    CONST robtarget p3347:= [[1487.1808479376136, -53.85036414256474, 992.500033578516], [0, 0, 1, 0], [0, 0, 0, 0], [9E9, 9E9, 9E9, 9E9, 9E9, 9E9]];
    CONST robtarget p3348:= [[1486.87587996053, -53.77743864899183, 992.500033578516], [0, 0, 1, 0], [0, 0, 0, 0], [9E9, 9E9, 9E9, 9E9, 9E9, 9E9]];
    CONST robtarget p3349:= [[1486.2803701551672, -53.64200512980345, 992.500033578516], [0, 0, 1, 0], [0, 0, 0, 0], [9E9, 9E9, 9E9, 9E9, 9E9, 9E9]];
    CONST robtarget p3350:= [[1486.1310585604317, -53.60921087716799, 992.500033578516], [0, 0, 1, 0], [0, 0, 0, 0], [9E9, 9E9, 9E9, 9E9, 9E9, 9E9]];
    CONST robtarget p3351:= [[1485.8708581653236, -53.549499191929584, 992.500033578516], [0, 0, 1, 0], [0, 0, 0, 0], [9E9, 9E9, 9E9, 9E9, 9E9, 9E9]];
    CONST robtarget p3352:= [[1485.4710135036546, -53.42288112586701, 992.500033578516], [0, 0, 1, 0], [0, 0, 0, 0], [9E9, 9E9, 9E9, 9E9, 9E9, 9E9]];
    CONST robtarget p3353:= [[1484.7300415279985, -53.201482726612156, 992.500033578516], [0, 0, 1, 0], [0, 0, 0, 0], [9E9, 9E9, 9E9, 9E9, 9E9, 9E9]];
    CONST robtarget p3354:= [[1484.6704427288005, -53.184901850971215, 992.500033578516], [0, 0, 1, 0], [0, 0, 0, 0], [9E9, 9E9, 9E9, 9E9, 9E9, 9E9]];
    CONST robtarget p3355:= [[1484.1819535099416, -53.02688255182427, 992.500033578516], [0, 0, 1, 0], [0, 0, 0, 0], [9E9, 9E9, 9E9, 9E9, 9E9, 9E9]];
    CONST robtarget p3356:= [[1483.924971929866, -52.957106793065265, 992.500033578516], [0, 0, 1, 0], [0, 0, 0, 0], [9E9, 9E9, 9E9, 9E9, 9E9, 9E9]];
    CONST robtarget p3357:= [[1483.840380212275, -52.9311047952195, 992.500033578516], [0, 0, 1, 0], [0, 0, 0, 0], [9E9, 9E9, 9E9, 9E9, 9E9, 9E9]];
    CONST robtarget p3358:= [[1483.1432899419212, -52.7309130716159, 992.500033578516], [0, 0, 1, 0], [0, 0, 0, 0], [9E9, 9E9, 9E9, 9E9, 9E9, 9E9]];
    CONST robtarget p3359:= [[1482.5943976643305, -52.5539516754126, 992.500033578516], [0, 0, 1, 0], [0, 0, 0, 0], [9E9, 9E9, 9E9, 9E9, 9E9, 9E9]];
    CONST robtarget p3360:= [[1482.3299474907458, -52.477779115658095, 992.500033578516], [0, 0, 1, 0], [0, 0, 0, 0], [9E9, 9E9, 9E9, 9E9, 9E9, 9E9]];
    CONST robtarget p3361:= [[1482.0010261741497, -52.38102058241606, 992.500033578516], [0, 0, 1, 0], [0, 0, 0, 0], [9E9, 9E9, 9E9, 9E9, 9E9, 9E9]];
    CONST robtarget p3362:= [[1481.5509158327018, -52.19874722975642, 992.500033578516], [0, 0, 1, 0], [0, 0, 0, 0], [9E9, 9E9, 9E9, 9E9, 9E9, 9E9]];
    CONST robtarget p3363:= [[1481.11315193246, -52.03041754687314, 992.500033578516], [0, 0, 1, 0], [0, 0, 0, 0], [9E9, 9E9, 9E9, 9E9, 9E9, 9E9]];
    CONST robtarget p3364:= [[1480.7938446633664, -51.90981571921251, 992.500033578516], [0, 0, 1, 0], [0, 0, 0, 0], [9E9, 9E9, 9E9, 9E9, 9E9, 9E9]];
    CONST robtarget p3365:= [[1480.54245378734, -51.821186668672595, 992.500033578516], [0, 0, 1, 0], [0, 0, 0, 0], [9E9, 9E9, 9E9, 9E9, 9E9, 9E9]];
    CONST robtarget p3366:= [[1480.41295095598, -51.770676335017384, 992.500033578516], [0, 0, 1, 0], [0, 0, 0, 0], [9E9, 9E9, 9E9, 9E9, 9E9, 9E9]];
    CONST robtarget p3367:= [[1480.1800345262973, -51.68403525234973, 992.500033578516], [0, 0, 1, 0], [0, 0, 0, 0], [9E9, 9E9, 9E9, 9E9, 9E9, 9E9]];
    CONST robtarget p3368:= [[1479.679579217019, -51.47045816045252, 992.500033578516], [0, 0, 1, 0], [0, 0, 0, 0], [9E9, 9E9, 9E9, 9E9, 9E9, 9E9]];
    CONST robtarget p3369:= [[1479.4242669133405, -51.37795854193503, 992.500033578516], [0, 0, 1, 0], [0, 0, 0, 0], [9E9, 9E9, 9E9, 9E9, 9E9, 9E9]];
    CONST robtarget p3370:= [[1479.11944210488, -51.27735123325023, 992.500033578516], [0, 0, 1, 0], [0, 0, 0, 0], [9E9, 9E9, 9E9, 9E9, 9E9, 9E9]];
    CONST robtarget p3371:= [[1478.9587402244965, -51.215634878753924, 992.500033578516], [0, 0, 1, 0], [0, 0, 0, 0], [9E9, 9E9, 9E9, 9E9, 9E9, 9E9]];
    CONST robtarget p3372:= [[1478.4078995703771, -51.00247068139136, 992.500033578516], [0, 0, 1, 0], [0, 0, 0, 0], [9E9, 9E9, 9E9, 9E9, 9E9, 9E9]];
    CONST robtarget p3373:= [[1477.9388565232143, -50.781502312677745, 992.500033578516], [0, 0, 1, 0], [0, 0, 0, 0], [9E9, 9E9, 9E9, 9E9, 9E9, 9E9]];
    CONST robtarget p3374:= [[1477.8276865064563, -50.735362270862616, 992.500033578516], [0, 0, 1, 0], [0, 0, 0, 0], [9E9, 9E9, 9E9, 9E9, 9E9, 9E9]];
    CONST robtarget p3375:= [[1477.1134991874192, -50.39257624403764, 992.500033578516], [0, 0, 1, 0], [0, 0, 0, 0], [9E9, 9E9, 9E9, 9E9, 9E9, 9E9]];
    CONST robtarget p3376:= [[1476.8127437004273, -50.25523619443268, 992.500033578516], [0, 0, 1, 0], [0, 0, 0, 0], [9E9, 9E9, 9E9, 9E9, 9E9, 9E9]];
    CONST robtarget p3377:= [[1476.581030580855, -50.14003244295683, 992.500033578516], [0, 0, 1, 0], [0, 0, 0, 0], [9E9, 9E9, 9E9, 9E9, 9E9, 9E9]];
    CONST robtarget p3378:= [[1476.2599962379181, -49.998280419195936, 992.500033578516], [0, 0, 1, 0], [0, 0, 0, 0], [9E9, 9E9, 9E9, 9E9, 9E9, 9E9]];
    CONST robtarget p3379:= [[1475.9104702559519, -49.840142555218655, 992.500033578516], [0, 0, 1, 0], [0, 0, 0, 0], [9E9, 9E9, 9E9, 9E9, 9E9, 9E9]];
    CONST robtarget p3380:= [[1475.4246393122305, -49.61222500336633, 992.500033578516], [0, 0, 1, 0], [0, 0, 0, 0], [9E9, 9E9, 9E9, 9E9, 9E9, 9E9]];
    CONST robtarget p3381:= [[1475.2041806503476, -49.49739674016412, 992.500033578516], [0, 0, 1, 0], [0, 0, 0, 0], [9E9, 9E9, 9E9, 9E9, 9E9, 9E9]];
    CONST robtarget p3382:= [[1474.6958711982638, -49.26805189035924, 992.500033578516], [0, 0, 1, 0], [0, 0, 0, 0], [9E9, 9E9, 9E9, 9E9, 9E9, 9E9]];
    CONST robtarget p3383:= [[1474.5346090707656, -49.18555260939496, 992.500033578516], [0, 0, 1, 0], [0, 0, 0, 0], [9E9, 9E9, 9E9, 9E9, 9E9, 9E9]];
    CONST robtarget p3384:= [[1474.4832461140786, -49.154293741446, 992.500033578516], [0, 0, 1, 0], [0, 0, 0, 0], [9E9, 9E9, 9E9, 9E9, 9E9, 9E9]];
    CONST robtarget p3385:= [[1473.9786661989287, -48.86779710482436, 992.500033578516], [0, 0, 1, 0], [0, 0, 0, 0], [9E9, 9E9, 9E9, 9E9, 9E9, 9E9]];
    CONST robtarget p3386:= [[1473.6783884368663, -48.684410713618966, 992.500033578516], [0, 0, 1, 0], [0, 0, 0, 0], [9E9, 9E9, 9E9, 9E9, 9E9, 9E9]];
    CONST robtarget p3387:= [[1473.4660175878853, -48.56892562768621, 992.500033578516], [0, 0, 1, 0], [0, 0, 0, 0], [9E9, 9E9, 9E9, 9E9, 9E9, 9E9]];
    CONST robtarget p3388:= [[1473.1610398384908, -48.40242427365542, 992.500033578516], [0, 0, 1, 0], [0, 0, 0, 0], [9E9, 9E9, 9E9, 9E9, 9E9, 9E9]];
    CONST robtarget p3389:= [[1472.8367985681707, -48.20621248412368, 992.500033578516], [0, 0, 1, 0], [0, 0, 0, 0], [9E9, 9E9, 9E9, 9E9, 9E9, 9E9]];
    CONST robtarget p3390:= [[1472.4561522390552, -48.009791772373376, 992.500033578516], [0, 0, 1, 0], [0, 0, 0, 0], [9E9, 9E9, 9E9, 9E9, 9E9, 9E9]];
    CONST robtarget p3391:= [[1472.1696380728436, -47.8383930113661, 992.500033578516], [0, 0, 1, 0], [0, 0, 0, 0], [9E9, 9E9, 9E9, 9E9, 9E9, 9E9]];
    CONST robtarget p3392:= [[1471.722110941695, -47.602916956820806, 992.500033578516], [0, 0, 1, 0], [0, 0, 0, 0], [9E9, 9E9, 9E9, 9E9, 9E9, 9E9]];
    CONST robtarget p3393:= [[1471.1098666991884, -47.258960245067954, 992.500033578516], [0, 0, 1, 0], [0, 0, 0, 0], [9E9, 9E9, 9E9, 9E9, 9E9, 9E9]];
    CONST robtarget p3394:= [[1470.720296694315, -47.00076007843536, 992.500033578516], [0, 0, 1, 0], [0, 0, 0, 0], [9E9, 9E9, 9E9, 9E9, 9E9, 9E9]];
    CONST robtarget p3395:= [[1470.35313472678, -46.74158028199264, 992.500033578516], [0, 0, 1, 0], [0, 0, 0, 0], [9E9, 9E9, 9E9, 9E9, 9E9, 9E9]];
    CONST robtarget p3396:= [[1470.1099347147267, -46.58885644915022, 992.500033578516], [0, 0, 1, 0], [0, 0, 0, 0], [9E9, 9E9, 9E9, 9E9, 9E9, 9E9]];
    CONST robtarget p3397:= [[1470.0533473815024, -46.55052435648606, 992.500033578516], [0, 0, 1, 0], [0, 0, 0, 0], [9E9, 9E9, 9E9, 9E9, 9E9, 9E9]];
    CONST robtarget p3398:= [[1469.7753241485486, -46.37599936065182, 992.500033578516], [0, 0, 1, 0], [0, 0, 0, 0], [9E9, 9E9, 9E9, 9E9, 9E9, 9E9]];
    CONST robtarget p3399:= [[1469.2259175939423, -46.010892422254685, 992.500033578516], [0, 0, 1, 0], [0, 0, 0, 0], [9E9, 9E9, 9E9, 9E9, 9E9, 9E9]];
    CONST robtarget p3400:= [[1468.7753752099943, -45.69106109718913, 992.500033578516], [0, 0, 1, 0], [0, 0, 0, 0], [9E9, 9E9, 9E9, 9E9, 9E9, 9E9]];
    CONST robtarget p3401:= [[1468.6198292044105, -45.59611312107232, 992.500033578516], [0, 0, 1, 0], [0, 0, 0, 0], [9E9, 9E9, 9E9, 9E9, 9E9, 9E9]];
    CONST robtarget p3402:= [[1468.0207049686155, -45.210283175710856, 992.500033578516], [0, 0, 1, 0], [0, 0, 0, 0], [9E9, 9E9, 9E9, 9E9, 9E9, 9E9]];
    CONST robtarget p3403:= [[1467.9426032268043, -45.16262396974101, 992.500033578516], [0, 0, 1, 0], [0, 0, 0, 0], [9E9, 9E9, 9E9, 9E9, 9E9, 9E9]];
    CONST robtarget p3404:= [[1467.7737235960665, -45.02594044699853, 992.500033578516], [0, 0, 1, 0], [0, 0, 0, 0], [9E9, 9E9, 9E9, 9E9, 9E9, 9E9]];
    CONST robtarget p3405:= [[1467.3306129242999, -44.708035159498436, 992.500033578516], [0, 0, 1, 0], [0, 0, 0, 0], [9E9, 9E9, 9E9, 9E9, 9E9, 9E9]];
    CONST robtarget p3406:= [[1466.7891375225997, -44.29104238444883, 992.500033578516], [0, 0, 1, 0], [0, 0, 0, 0], [9E9, 9E9, 9E9, 9E9, 9E9, 9E9]];
    CONST robtarget p3407:= [[1466.6930449917838, -44.218374738723874, 992.500033578516], [0, 0, 1, 0], [0, 0, 0, 0], [9E9, 9E9, 9E9, 9E9, 9E9, 9E9]];
    CONST robtarget p3408:= [[1466.6125504698477, -44.15573091450402, 992.500033578516], [0, 0, 1, 0], [0, 0, 0, 0], [9E9, 9E9, 9E9, 9E9, 9E9, 9E9]];
    CONST robtarget p3409:= [[1466.5453531413737, -44.1016987432777, 992.500033578516], [0, 0, 1, 0], [0, 0, 0, 0], [9E9, 9E9, 9E9, 9E9, 9E9, 9E9]];
    CONST robtarget p3410:= [[1466.0727069489167, -43.73594157482748, 992.500033578516], [0, 0, 1, 0], [0, 0, 0, 0], [9E9, 9E9, 9E9, 9E9, 9E9, 9E9]];
    CONST robtarget p3411:= [[1465.8449401864993, -43.55418955615802, 992.500033578516], [0, 0, 1, 0], [0, 0, 0, 0], [9E9, 9E9, 9E9, 9E9, 9E9, 9E9]];
    CONST robtarget p3412:= [[1465.4027049879091, -43.170989150472266, 992.500033578516], [0, 0, 1, 0], [0, 0, 0, 0], [9E9, 9E9, 9E9, 9E9, 9E9, 9E9]];
    CONST robtarget p3413:= [[1465.0737708983593, -42.91529482758523, 992.500033578516], [0, 0, 1, 0], [0, 0, 0, 0], [9E9, 9E9, 9E9, 9E9, 9E9, 9E9]];
    CONST robtarget p3414:= [[1464.758462542708, -42.69398236756925, 992.500033578516], [0, 0, 1, 0], [0, 0, 0, 0], [9E9, 9E9, 9E9, 9E9, 9E9, 9E9]];
    CONST robtarget p3415:= [[1464.7064575827471, -42.64949993988721, 992.500033578516], [0, 0, 1, 0], [0, 0, 0, 0], [9E9, 9E9, 9E9, 9E9, 9E9, 9E9]];
    CONST robtarget p3416:= [[1464.2049615544438, -42.25132751961473, 992.500033578516], [0, 0, 1, 0], [0, 0, 0, 0], [9E9, 9E9, 9E9, 9E9, 9E9, 9E9]];
    CONST robtarget p3417:= [[1463.630038306874, -41.732635097727126, 992.500033578516], [0, 0, 1, 0], [0, 0, 0, 0], [9E9, 9E9, 9E9, 9E9, 9E9, 9E9]];
    CONST robtarget p3418:= [[1463.4169508414868, -41.54373278258235, 992.500033578516], [0, 0, 1, 0], [0, 0, 0, 0], [9E9, 9E9, 9E9, 9E9, 9E9, 9E9]];
    CONST robtarget p3419:= [[1462.9378345294456, -41.10845872936408, 992.500033578516], [0, 0, 1, 0], [0, 0, 0, 0], [9E9, 9E9, 9E9, 9E9, 9E9, 9E9]];
    CONST robtarget p3420:= [[1462.7967031838916, -40.970170988054306, 992.500033578516], [0, 0, 1, 0], [0, 0, 0, 0], [9E9, 9E9, 9E9, 9E9, 9E9, 9E9]];
    CONST robtarget p3421:= [[1462.3892181115343, -40.624094337487456, 992.500033578516], [0, 0, 1, 0], [0, 0, 0, 0], [9E9, 9E9, 9E9, 9E9, 9E9, 9E9]];
    CONST robtarget p3422:= [[1462.1484926621697, -40.40265536007567, 992.500033578516], [0, 0, 1, 0], [0, 0, 0, 0], [9E9, 9E9, 9E9, 9E9, 9E9, 9E9]];
    CONST robtarget p3423:= [[1461.9188144316706, -40.19832888780002, 992.500033578516], [0, 0, 1, 0], [0, 0, 0, 0], [9E9, 9E9, 9E9, 9E9, 9E9, 9E9]];
    CONST robtarget p3424:= [[1461.7316067411623, -40.03100624215904, 992.500033578516], [0, 0, 1, 0], [0, 0, 0, 0], [9E9, 9E9, 9E9, 9E9, 9E9, 9E9]];
    CONST robtarget p3425:= [[1461.255703154484, -39.54403407148257, 992.500033578516], [0, 0, 1, 0], [0, 0, 0, 0], [9E9, 9E9, 9E9, 9E9, 9E9, 9E9]];
    CONST robtarget p3426:= [[1461.113593493523, -39.417810138225164, 992.500033578516], [0, 0, 1, 0], [0, 0, 0, 0], [9E9, 9E9, 9E9, 9E9, 9E9, 9E9]];
    CONST robtarget p3427:= [[1460.8243082681377, -39.117556858200075, 992.500033578516], [0, 0, 1, 0], [0, 0, 0, 0], [9E9, 9E9, 9E9, 9E9, 9E9, 9E9]];
    CONST robtarget p3428:= [[1460.6515882379688, -38.94266158745661, 992.500033578516], [0, 0, 1, 0], [0, 0, 0, 0], [9E9, 9E9, 9E9, 9E9, 9E9, 9E9]];
    CONST robtarget p3429:= [[1460.2690854199782, -38.52851516353172, 992.500033578516], [0, 0, 1, 0], [0, 0, 0, 0], [9E9, 9E9, 9E9, 9E9, 9E9, 9E9]];
    CONST robtarget p3430:= [[1460.145444752096, -38.401242774626866, 992.500033578516], [0, 0, 1, 0], [0, 0, 0, 0], [9E9, 9E9, 9E9, 9E9, 9E9, 9E9]];
    CONST robtarget p3431:= [[1459.9006997120866, -38.164320817301046, 992.500033578516], [0, 0, 1, 0], [0, 0, 0, 0], [9E9, 9E9, 9E9, 9E9, 9E9, 9E9]];
    CONST robtarget p3432:= [[1459.3337364708455, -37.572283003185476, 992.500033578516], [0, 0, 1, 0], [0, 0, 0, 0], [9E9, 9E9, 9E9, 9E9, 9E9, 9E9]];
    CONST robtarget p3433:= [[1459.0295125348634, -37.25995643815945, 992.500033578516], [0, 0, 1, 0], [0, 0, 0, 0], [9E9, 9E9, 9E9, 9E9, 9E9, 9E9]];
    CONST robtarget p3434:= [[1458.8623888247864, -37.06729815014819, 992.500033578516], [0, 0, 1, 0], [0, 0, 0, 0], [9E9, 9E9, 9E9, 9E9, 9E9, 9E9]];
    CONST robtarget p3435:= [[1458.6325053445294, -36.82857891687241, 992.500033578516], [0, 0, 1, 0], [0, 0, 0, 0], [9E9, 9E9, 9E9, 9E9, 9E9, 9E9]];
    CONST robtarget p3436:= [[1458.2543383331513, -36.37668611510166, 992.500033578516], [0, 0, 1, 0], [0, 0, 0, 0], [9E9, 9E9, 9E9, 9E9, 9E9, 9E9]];
    CONST robtarget p3437:= [[1458.027121084747, -36.0990363969632, 992.500033578516], [0, 0, 1, 0], [0, 0, 0, 0], [9E9, 9E9, 9E9, 9E9, 9E9, 9E9]];
    CONST robtarget p3438:= [[1457.606983168909, -35.57616256060792, 992.500033578516], [0, 0, 1, 0], [0, 0, 0, 0], [9E9, 9E9, 9E9, 9E9, 9E9, 9E9]];
    CONST robtarget p3439:= [[1457.4283569201107, -35.37977836110465, 992.500033578516], [0, 0, 1, 0], [0, 0, 0, 0], [9E9, 9E9, 9E9, 9E9, 9E9, 9E9]];
    CONST robtarget p3440:= [[1457.3011215960366, -35.219036477829, 992.500033578516], [0, 0, 1, 0], [0, 0, 0, 0], [9E9, 9E9, 9E9, 9E9, 9E9, 9E9]];
    CONST robtarget p3441:= [[1456.9818584121829, -34.82149399107248, 992.500033578516], [0, 0, 1, 0], [0, 0, 0, 0], [9E9, 9E9, 9E9, 9E9, 9E9, 9E9]];
    CONST robtarget p3442:= [[1456.6636166327598, -34.45580181917994, 992.500033578516], [0, 0, 1, 0], [0, 0, 0, 0], [9E9, 9E9, 9E9, 9E9, 9E9, 9E9]];
    CONST robtarget p3443:= [[1456.5323695679463, -34.29554978453682, 992.500033578516], [0, 0, 1, 0], [0, 0, 0, 0], [9E9, 9E9, 9E9, 9E9, 9E9, 9E9]];
    CONST robtarget p3444:= [[1456.3233257777242, -34.045472209657945, 992.500033578516], [0, 0, 1, 0], [0, 0, 0, 0], [9E9, 9E9, 9E9, 9E9, 9E9, 9E9]];
    CONST robtarget p3445:= [[1456.2166850399808, -33.918669267549404, 992.500033578516], [0, 0, 1, 0], [0, 0, 0, 0], [9E9, 9E9, 9E9, 9E9, 9E9, 9E9]];
    CONST robtarget p3446:= [[1456.0384938500167, -33.6602158090042, 992.500033578516], [0, 0, 1, 0], [0, 0, 0, 0], [9E9, 9E9, 9E9, 9E9, 9E9, 9E9]];
    CONST robtarget p3447:= [[1455.6908502470403, -33.169738455154864, 992.500033578516], [0, 0, 1, 0], [0, 0, 0, 0], [9E9, 9E9, 9E9, 9E9, 9E9, 9E9]];
    CONST robtarget p3448:= [[1455.5760633333898, -33.019124983816305, 992.500033578516], [0, 0, 1, 0], [0, 0, 0, 0], [9E9, 9E9, 9E9, 9E9, 9E9, 9E9]];
    CONST robtarget p3449:= [[1455.4907916846773, -32.91439129744002, 992.500033578516], [0, 0, 1, 0], [0, 0, 0, 0], [9E9, 9E9, 9E9, 9E9, 9E9, 9E9]];
    CONST robtarget p3450:= [[1455.3933901197092, -32.7724652494033, 992.500033578516], [0, 0, 1, 0], [0, 0, 0, 0], [9E9, 9E9, 9E9, 9E9, 9E9, 9E9]];
    CONST robtarget p3451:= [[1455.0836451860825, -32.34474490769912, 992.500033578516], [0, 0, 1, 0], [0, 0, 0, 0], [9E9, 9E9, 9E9, 9E9, 9E9, 9E9]];
    CONST robtarget p3452:= [[1455.0256362747637, -32.27203612221187, 992.500033578516], [0, 0, 1, 0], [0, 0, 0, 0], [9E9, 9E9, 9E9, 9E9, 9E9, 9E9]];
    CONST robtarget p3453:= [[1454.9849089470888, -32.20635720096585, 992.500033578516], [0, 0, 1, 0], [0, 0, 0, 0], [9E9, 9E9, 9E9, 9E9, 9E9, 9E9]];
    CONST robtarget p3454:= [[1454.8265637840655, -31.96721797953569, 992.500033578516], [0, 0, 1, 0], [0, 0, 0, 0], [9E9, 9E9, 9E9, 9E9, 9E9, 9E9]];
    CONST robtarget p3455:= [[1454.6476826405483, -31.70587733425765, 992.500033578516], [0, 0, 1, 0], [0, 0, 0, 0], [9E9, 9E9, 9E9, 9E9, 9E9, 9E9]];
    CONST robtarget p3456:= [[1454.2879280135612, -31.233368738334782, 992.500033578516], [0, 0, 1, 0], [0, 0, 0, 0], [9E9, 9E9, 9E9, 9E9, 9E9, 9E9]];
    CONST robtarget p3457:= [[1454.2310540800454, -31.15991131192105, 992.500033578516], [0, 0, 1, 0], [0, 0, 0, 0], [9E9, 9E9, 9E9, 9E9, 9E9, 9E9]];
    CONST robtarget p3458:= [[1454.0148081812833, -30.85863960132579, 992.500033578516], [0, 0, 1, 0], [0, 0, 0, 0], [9E9, 9E9, 9E9, 9E9, 9E9, 9E9]];
    CONST robtarget p3459:= [[1453.8782259279728, -30.658488528819916, 992.500033578516], [0, 0, 1, 0], [0, 0, 0, 0], [9E9, 9E9, 9E9, 9E9, 9E9, 9E9]];
    CONST robtarget p3460:= [[1453.7047332343661, -30.39940063569474, 992.500033578516], [0, 0, 1, 0], [0, 0, 0, 0], [9E9, 9E9, 9E9, 9E9, 9E9, 9E9]];
    CONST robtarget p3461:= [[1453.3569685886248, -29.82367260534658, 992.500033578516], [0, 0, 1, 0], [0, 0, 0, 0], [9E9, 9E9, 9E9, 9E9, 9E9, 9E9]];
    CONST robtarget p3462:= [[1453.1568211893682, -29.49263065365509, 992.500033578516], [0, 0, 1, 0], [0, 0, 0, 0], [9E9, 9E9, 9E9, 9E9, 9E9, 9E9]];
    CONST robtarget p3463:= [[1452.998690278866, -29.238377319886283, 992.500033578516], [0, 0, 1, 0], [0, 0, 0, 0], [9E9, 9E9, 9E9, 9E9, 9E9, 9E9]];
    CONST robtarget p3464:= [[1452.8914361103687, -29.0719103079496, 992.500033578516], [0, 0, 1, 0], [0, 0, 0, 0], [9E9, 9E9, 9E9, 9E9, 9E9, 9E9]];
    CONST robtarget p3465:= [[1452.710971989498, -28.76624786149432, 992.500033578516], [0, 0, 1, 0], [0, 0, 0, 0], [9E9, 9E9, 9E9, 9E9, 9E9, 9E9]];
    CONST robtarget p3466:= [[1452.4950323117525, -28.415016794012246, 992.500033578516], [0, 0, 1, 0], [0, 0, 0, 0], [9E9, 9E9, 9E9, 9E9, 9E9, 9E9]];
    CONST robtarget p3467:= [[1452.3180448544556, -28.09806084352619, 992.500033578516], [0, 0, 1, 0], [0, 0, 0, 0], [9E9, 9E9, 9E9, 9E9, 9E9, 9E9]];
    CONST robtarget p3468:= [[1452.0877233748438, -27.75046800727705, 992.500033578516], [0, 0, 1, 0], [0, 0, 0, 0], [9E9, 9E9, 9E9, 9E9, 9E9, 9E9]];
    CONST robtarget p3469:= [[1451.6606058467132, -27.04640524100038, 992.500033578516], [0, 0, 1, 0], [0, 0, 0, 0], [9E9, 9E9, 9E9, 9E9, 9E9, 9E9]];
    CONST robtarget p3470:= [[1451.5962239303992, -26.91805172162867, 992.500033578516], [0, 0, 1, 0], [0, 0, 0, 0], [9E9, 9E9, 9E9, 9E9, 9E9, 9E9]];
    CONST robtarget p3471:= [[1451.3722419824685, -26.459298942251095, 992.500033578516], [0, 0, 1, 0], [0, 0, 0, 0], [9E9, 9E9, 9E9, 9E9, 9E9, 9E9]];
    CONST robtarget p3472:= [[1451.218050210988, -26.183150546714593, 992.500033578516], [0, 0, 1, 0], [0, 0, 0, 0], [9E9, 9E9, 9E9, 9E9, 9E9, 9E9]];
    CONST robtarget p3473:= [[1451.0414892764409, -25.833096766525777, 992.500033578516], [0, 0, 1, 0], [0, 0, 0, 0], [9E9, 9E9, 9E9, 9E9, 9E9, 9E9]];
    CONST robtarget p3474:= [[1450.937388649569, -25.626608472575832, 992.500033578516], [0, 0, 1, 0], [0, 0, 0, 0], [9E9, 9E9, 9E9, 9E9, 9E9, 9E9]];
    CONST robtarget p3475:= [[1450.7626135189141, -25.29657327285075, 992.500033578516], [0, 0, 1, 0], [0, 0, 0, 0], [9E9, 9E9, 9E9, 9E9, 9E9, 9E9]];
    CONST robtarget p3476:= [[1450.5767888187597, -24.931814257633114, 992.500033578516], [0, 0, 1, 0], [0, 0, 0, 0], [9E9, 9E9, 9E9, 9E9, 9E9, 9E9]];
    CONST robtarget p3477:= [[1450.3107905505367, -24.420648005814748, 992.500033578516], [0, 0, 1, 0], [0, 0, 0, 0], [9E9, 9E9, 9E9, 9E9, 9E9, 9E9]];
    CONST robtarget p3478:= [[1450.0703210397674, -23.92574279306882, 992.500033578516], [0, 0, 1, 0], [0, 0, 0, 0], [9E9, 9E9, 9E9, 9E9, 9E9, 9E9]];
    CONST robtarget p3479:= [[1449.8480002303459, -23.493559697346946, 992.500033578516], [0, 0, 1, 0], [0, 0, 0, 0], [9E9, 9E9, 9E9, 9E9, 9E9, 9E9]];
    CONST robtarget p3480:= [[1449.8401476031047, -23.47896840986204, 992.500033578516], [0, 0, 1, 0], [0, 0, 0, 0], [9E9, 9E9, 9E9, 9E9, 9E9, 9E9]];
    CONST robtarget p3481:= [[1449.7743196513866, -23.329523112877595, 992.500033578516], [0, 0, 1, 0], [0, 0, 0, 0], [9E9, 9E9, 9E9, 9E9, 9E9, 9E9]];
    CONST robtarget p3482:= [[1449.490067459615, -22.636335832590113, 992.500033578516], [0, 0, 1, 0], [0, 0, 0, 0], [9E9, 9E9, 9E9, 9E9, 9E9, 9E9]];
    CONST robtarget p3483:= [[1449.3793270596516, -22.352133946995814, 992.500033578516], [0, 0, 1, 0], [0, 0, 0, 0], [9E9, 9E9, 9E9, 9E9, 9E9, 9E9]];
    CONST robtarget p3484:= [[1449.1617233913162, -21.89352333667363, 992.500033578516], [0, 0, 1, 0], [0, 0, 0, 0], [9E9, 9E9, 9E9, 9E9, 9E9, 9E9]];
    CONST robtarget p3485:= [[1449.1176045895998, -21.798337941021806, 992.500033578516], [0, 0, 1, 0], [0, 0, 0, 0], [9E9, 9E9, 9E9, 9E9, 9E9, 9E9]];
    CONST robtarget p3486:= [[1448.9987091221262, -21.52112647747648, 992.500033578516], [0, 0, 1, 0], [0, 0, 0, 0], [9E9, 9E9, 9E9, 9E9, 9E9, 9E9]];
    CONST robtarget p3487:= [[1448.9425986005542, -21.376342990196108, 992.500033578516], [0, 0, 1, 0], [0, 0, 0, 0], [9E9, 9E9, 9E9, 9E9, 9E9, 9E9]];
    CONST robtarget p3488:= [[1448.8290224991424, -21.113528522465906, 992.500033578516], [0, 0, 1, 0], [0, 0, 0, 0], [9E9, 9E9, 9E9, 9E9, 9E9, 9E9]];
    CONST robtarget p3489:= [[1448.7250837405568, -20.880642118370204, 992.500033578516], [0, 0, 1, 0], [0, 0, 0, 0], [9E9, 9E9, 9E9, 9E9, 9E9, 9E9]];
    CONST robtarget p3490:= [[1448.592786106188, -20.552964563670386, 992.500033578516], [0, 0, 1, 0], [0, 0, 0, 0], [9E9, 9E9, 9E9, 9E9, 9E9, 9E9]];
    CONST robtarget p3491:= [[1448.4839737748262, -20.304959229817023, 992.500033578516], [0, 0, 1, 0], [0, 0, 0, 0], [9E9, 9E9, 9E9, 9E9, 9E9, 9E9]];
    CONST robtarget p3492:= [[1448.4351233271393, -20.17234874689011, 992.500033578516], [0, 0, 1, 0], [0, 0, 0, 0], [9E9, 9E9, 9E9, 9E9, 9E9, 9E9]];
    CONST robtarget p3493:= [[1448.365696399131, -19.988516313687505, 992.500033578516], [0, 0, 1, 0], [0, 0, 0, 0], [9E9, 9E9, 9E9, 9E9, 9E9, 9E9]];
    CONST robtarget p3494:= [[1448.2067766799746, -19.62882008426967, 992.500033578516], [0, 0, 1, 0], [0, 0, 0, 0], [9E9, 9E9, 9E9, 9E9, 9E9, 9E9]];
    CONST robtarget p3495:= [[1448.1445776164344, -19.4193974113416, 992.500033578516], [0, 0, 1, 0], [0, 0, 0, 0], [9E9, 9E9, 9E9, 9E9, 9E9, 9E9]];
    CONST robtarget p3496:= [[1448.0330998698576, -19.101623794848415, 992.500033578516], [0, 0, 1, 0], [0, 0, 0, 0], [9E9, 9E9, 9E9, 9E9, 9E9, 9E9]];
    CONST robtarget p3497:= [[1447.99477449825, -18.9666175903102, 992.500033578516], [0, 0, 1, 0], [0, 0, 0, 0], [9E9, 9E9, 9E9, 9E9, 9E9, 9E9]];
    CONST robtarget p3498:= [[1447.8493306377272, -18.50273578183046, 992.500033578516], [0, 0, 1, 0], [0, 0, 0, 0], [9E9, 9E9, 9E9, 9E9, 9E9, 9E9]];
    CONST robtarget p3499:= [[1447.710091458263, -18.152457475056202, 992.500033578516], [0, 0, 1, 0], [0, 0, 0, 0], [9E9, 9E9, 9E9, 9E9, 9E9, 9E9]];
    CONST robtarget p3500:= [[1447.6300222279517, -17.927275169957845, 992.500033578516], [0, 0, 1, 0], [0, 0, 0, 0], [9E9, 9E9, 9E9, 9E9, 9E9, 9E9]];
    CONST robtarget p3501:= [[1447.4531103531453, -17.39982928374014, 992.500033578516], [0, 0, 1, 0], [0, 0, 0, 0], [9E9, 9E9, 9E9, 9E9, 9E9, 9E9]];
    CONST robtarget p3502:= [[1447.290968872516, -16.935627813711996, 992.500033578516], [0, 0, 1, 0], [0, 0, 0, 0], [9E9, 9E9, 9E9, 9E9, 9E9, 9E9]];
    CONST robtarget p3503:= [[1447.1409217422781, -16.490624161224908, 992.500033578516], [0, 0, 1, 0], [0, 0, 0, 0], [9E9, 9E9, 9E9, 9E9, 9E9, 9E9]];
    CONST robtarget p3504:= [[1447.1016279657379, -16.37617355106139, 992.500033578516], [0, 0, 1, 0], [0, 0, 0, 0], [9E9, 9E9, 9E9, 9E9, 9E9, 9E9]];
    CONST robtarget p3505:= [[1446.9486445579141, -15.93663314206443, 992.500033578516], [0, 0, 1, 0], [0, 0, 0, 0], [9E9, 9E9, 9E9, 9E9, 9E9, 9E9]];
    CONST robtarget p3506:= [[1446.8152564865, -15.401278346021833, 992.500033578516], [0, 0, 1, 0], [0, 0, 0, 0], [9E9, 9E9, 9E9, 9E9, 9E9, 9E9]];
    CONST robtarget p3507:= [[1446.7295768237227, -15.011047130391788, 992.500033578516], [0, 0, 1, 0], [0, 0, 0, 0], [9E9, 9E9, 9E9, 9E9, 9E9, 9E9]];
    CONST robtarget p3508:= [[1446.612030653954, -14.612522235073065, 992.500033578516], [0, 0, 1, 0], [0, 0, 0, 0], [9E9, 9E9, 9E9, 9E9, 9E9, 9E9]];
    CONST robtarget p3509:= [[1446.562436568088, -14.409856126046947, 992.500033578516], [0, 0, 1, 0], [0, 0, 0, 0], [9E9, 9E9, 9E9, 9E9, 9E9, 9E9]];
    CONST robtarget p3510:= [[1446.4816306006028, -14.123993635031042, 992.500033578516], [0, 0, 1, 0], [0, 0, 0, 0], [9E9, 9E9, 9E9, 9E9, 9E9, 9E9]];
    CONST robtarget p3511:= [[1446.4024648372183, -13.82132106732427, 992.500033578516], [0, 0, 1, 0], [0, 0, 0, 0], [9E9, 9E9, 9E9, 9E9, 9E9, 9E9]];
    CONST robtarget p3512:= [[1446.2581467404725, -13.273706195437228, 992.500033578516], [0, 0, 1, 0], [0, 0, 0, 0], [9E9, 9E9, 9E9, 9E9, 9E9, 9E9]];
    CONST robtarget p3513:= [[1446.138194338032, -12.802805213387018, 992.500033578516], [0, 0, 1, 0], [0, 0, 0, 0], [9E9, 9E9, 9E9, 9E9, 9E9, 9E9]];
    CONST robtarget p3514:= [[1445.938513046241, -12.033124951805334, 992.500033578516], [0, 0, 1, 0], [0, 0, 0, 0], [9E9, 9E9, 9E9, 9E9, 9E9, 9E9]];
    CONST robtarget p3515:= [[1445.923760106864, -11.954278447784198, 992.500033578516], [0, 0, 1, 0], [0, 0, 0, 0], [9E9, 9E9, 9E9, 9E9, 9E9, 9E9]];
    CONST robtarget p3516:= [[1445.8823964391556, -11.699978278644252, 992.500033578516], [0, 0, 1, 0], [0, 0, 0, 0], [9E9, 9E9, 9E9, 9E9, 9E9, 9E9]];
    CONST robtarget p3517:= [[1445.858249235026, -11.56425325097375, 992.500033578516], [0, 0, 1, 0], [0, 0, 0, 0], [9E9, 9E9, 9E9, 9E9, 9E9, 9E9]];
    CONST robtarget p3518:= [[1445.8403405666065, -11.471894054016317, 992.500033578516], [0, 0, 1, 0], [0, 0, 0, 0], [9E9, 9E9, 9E9, 9E9, 9E9, 9E9]];
    CONST robtarget p3519:= [[1445.8119897791105, -11.31890541957739, 992.500033578516], [0, 0, 1, 0], [0, 0, 0, 0], [9E9, 9E9, 9E9, 9E9, 9E9, 9E9]];
    CONST robtarget p3520:= [[1445.6586432752847, -10.571474974941466, 992.500033578516], [0, 0, 1, 0], [0, 0, 0, 0], [9E9, 9E9, 9E9, 9E9, 9E9, 9E9]];
    CONST robtarget p3521:= [[1445.6416589634534, -10.469936371774459, 992.500033578516], [0, 0, 1, 0], [0, 0, 0, 0], [9E9, 9E9, 9E9, 9E9, 9E9, 9E9]];
    CONST robtarget p3522:= [[1445.593108080078, -10.181225910298949, 992.500033578516], [0, 0, 1, 0], [0, 0, 0, 0], [9E9, 9E9, 9E9, 9E9, 9E9, 9E9]];
    CONST robtarget p3523:= [[1445.5468631117226, -9.94266718882993, 992.500033578516], [0, 0, 1, 0], [0, 0, 0, 0], [9E9, 9E9, 9E9, 9E9, 9E9, 9E9]];
    CONST robtarget p3524:= [[1445.4547342362575, -9.444153894284227, 992.500033578516], [0, 0, 1, 0], [0, 0, 0, 0], [9E9, 9E9, 9E9, 9E9, 9E9, 9E9]];
    CONST robtarget p3525:= [[1445.3714447736427, -9.010887898255525, 992.500033578516], [0, 0, 1, 0], [0, 0, 0, 0], [9E9, 9E9, 9E9, 9E9, 9E9, 9E9]];
    CONST robtarget p3526:= [[1445.2732767246098, -8.483335926873181, 992.500033578516], [0, 0, 1, 0], [0, 0, 0, 0], [9E9, 9E9, 9E9, 9E9, 9E9, 9E9]];
    CONST robtarget p3527:= [[1445.25313275983, -8.374357104724801, 992.500033578516], [0, 0, 1, 0], [0, 0, 0, 0], [9E9, 9E9, 9E9, 9E9, 9E9, 9E9]];
    CONST robtarget p3528:= [[1445.2095806999887, -7.978981630061071, 992.500033578516], [0, 0, 1, 0], [0, 0, 0, 0], [9E9, 9E9, 9E9, 9E9, 9E9, 9E9]];
    CONST robtarget p3529:= [[1445.1256311191448, -7.365424011079028, 992.500033578516], [0, 0, 1, 0], [0, 0, 0, 0], [9E9, 9E9, 9E9, 9E9, 9E9, 9E9]];
    CONST robtarget p3530:= [[1445.093389233748, -7.0807262688907, 992.500033578516], [0, 0, 1, 0], [0, 0, 0, 0], [9E9, 9E9, 9E9, 9E9, 9E9, 9E9]];
    CONST robtarget p3531:= [[1445.0770091126997, -6.938185816370513, 992.500033578516], [0, 0, 1, 0], [0, 0, 0, 0], [9E9, 9E9, 9E9, 9E9, 9E9, 9E9]];
    CONST robtarget p3532:= [[1445.0262101714134, -6.493044737196186, 992.500033578516], [0, 0, 1, 0], [0, 0, 0, 0], [9E9, 9E9, 9E9, 9E9, 9E9, 9E9]];
    CONST robtarget p3533:= [[1444.9589223996718, -5.8520673038310775, 992.500033578516], [0, 0, 1, 0], [0, 0, 0, 0], [9E9, 9E9, 9E9, 9E9, 9E9, 9E9]];
    CONST robtarget p3534:= [[1444.942957200915, -5.661944186401996, 992.500033578516], [0, 0, 1, 0], [0, 0, 0, 0], [9E9, 9E9, 9E9, 9E9, 9E9, 9E9]];
    CONST robtarget p3535:= [[1444.93858482627, -5.619251634791567, 992.500033578516], [0, 0, 1, 0], [0, 0, 0, 0], [9E9, 9E9, 9E9, 9E9, 9E9, 9E9]];
    CONST robtarget p3536:= [[1444.8754307775705, -5.054964641155507, 992.500033578516], [0, 0, 1, 0], [0, 0, 0, 0], [9E9, 9E9, 9E9, 9E9, 9E9, 9E9]];
    CONST robtarget p3537:= [[1444.8299077384686, -4.715481991021605, 992.500033578516], [0, 0, 1, 0], [0, 0, 0, 0], [9E9, 9E9, 9E9, 9E9, 9E9, 9E9]];
    CONST robtarget p3538:= [[1444.8149547608155, -4.59749911617368, 992.500033578516], [0, 0, 1, 0], [0, 0, 0, 0], [9E9, 9E9, 9E9, 9E9, 9E9, 9E9]];
    CONST robtarget p3539:= [[1444.813428207593, -4.551174813249077, 992.500033578516], [0, 0, 1, 0], [0, 0, 0, 0], [9E9, 9E9, 9E9, 9E9, 9E9, 9E9]];
    CONST robtarget p3540:= [[1444.789642708461, -4.073721118029198, 992.500033578516], [0, 0, 1, 0], [0, 0, 0, 0], [9E9, 9E9, 9E9, 9E9, 9E9, 9E9]];
    CONST robtarget p3541:= [[1444.7565988447466, -3.8072675157633995, 992.500033578516], [0, 0, 1, 0], [0, 0, 0, 0], [9E9, 9E9, 9E9, 9E9, 9E9, 9E9]];
    CONST robtarget p3542:= [[1444.7290518154543, -3.3100920942163583, 992.500033578516], [0, 0, 1, 0], [0, 0, 0, 0], [9E9, 9E9, 9E9, 9E9, 9E9, 9E9]];
    CONST robtarget p3543:= [[1444.7199692749316, -2.7495599834710163, 992.500033578516], [0, 0, 1, 0], [0, 0, 0, 0], [9E9, 9E9, 9E9, 9E9, 9E9, 9E9]];
    CONST robtarget p3544:= [[1444.719868805816, -2.621050148635959, 992.500033578516], [0, 0, 1, 0], [0, 0, 0, 0], [9E9, 9E9, 9E9, 9E9, 9E9, 9E9]];
    CONST robtarget p3545:= [[1444.7158211593426, -2.3672287977827295, 992.500033578516], [0, 0, 1, 0], [0, 0, 0, 0], [9E9, 9E9, 9E9, 9E9, 9E9, 9E9]];
    CONST robtarget p3546:= [[1444.4663405446136, -2.5286384905235195, 993.500033578516], [0, 0, 1, 0], [0, 0, 0, 0], [9E9, 9E9, 9E9, 9E9, 9E9, 9E9]];
    CONST robtarget p3547:= [[1444.4441635007622, -1.8292304588618151, 993.500033578516], [0, 0, 1, 0], [0, 0, 0, 0], [9E9, 9E9, 9E9, 9E9, 9E9, 9E9]];
    CONST robtarget p3548:= [[1444.428525603863, -1.3479255931139704, 993.500033578516], [0, 0, 1, 0], [0, 0, 0, 0], [9E9, 9E9, 9E9, 9E9, 9E9, 9E9]];
    CONST robtarget p3549:= [[1444.4174000410437, -1.0475235956110112, 993.500033578516], [0, 0, 1, 0], [0, 0, 0, 0], [9E9, 9E9, 9E9, 9E9, 9E9, 9E9]];
    CONST robtarget p3550:= [[1444.4104387675868, -0.7931788061941205, 993.500033578516], [0, 0, 1, 0], [0, 0, 0, 0], [9E9, 9E9, 9E9, 9E9, 9E9, 9E9]];
    CONST robtarget p3551:= [[1444.3908201907582, -0.5000305658536632, 993.500033578516], [0, 0, 1, 0], [0, 0, 0, 0], [9E9, 9E9, 9E9, 9E9, 9E9, 9E9]];
    CONST robtarget p3552:= [[1444.3878403243452, -0.4057105965694774, 993.500033578516], [0, 0, 1, 0], [0, 0, 0, 0], [9E9, 9E9, 9E9, 9E9, 9E9, 9E9]];
    CONST robtarget p3553:= [[1444.378812719543, 0.04115573668573802, 993.500033578516], [0, 0, 1, 0], [0, 0, 0, 0], [9E9, 9E9, 9E9, 9E9, 9E9, 9E9]];
    CONST robtarget p3554:= [[1444.3971996529272, 0.7206241421897772, 993.500033578516], [0, 0, 1, 0], [0, 0, 0, 0], [9E9, 9E9, 9E9, 9E9, 9E9, 9E9]];
    CONST robtarget p3555:= [[1444.4477772540863, 1.2756732553033174, 993.500033578516], [0, 0, 1, 0], [0, 0, 0, 0], [9E9, 9E9, 9E9, 9E9, 9E9, 9E9]];
    CONST robtarget p3556:= [[1444.470766942313, 1.6320465733553675, 993.500033578516], [0, 0, 1, 0], [0, 0, 0, 0], [9E9, 9E9, 9E9, 9E9, 9E9, 9E9]];
    CONST robtarget p3557:= [[1444.4563950861611, 2.3975781072703626, 993.500033578516], [0, 0, 1, 0], [0, 0, 0, 0], [9E9, 9E9, 9E9, 9E9, 9E9, 9E9]];
    CONST robtarget p3558:= [[1444.4969997494484, 3.4595933898866207, 993.500033578516], [0, 0, 1, 0], [0, 0, 0, 0], [9E9, 9E9, 9E9, 9E9, 9E9, 9E9]];
    CONST robtarget p3559:= [[1444.5180270622116, 3.9283626343067226, 993.500033578516], [0, 0, 1, 0], [0, 0, 0, 0], [9E9, 9E9, 9E9, 9E9, 9E9, 9E9]];
    CONST robtarget p3560:= [[1444.5320755007199, 4.180217495226117, 993.500033578516], [0, 0, 1, 0], [0, 0, 0, 0], [9E9, 9E9, 9E9, 9E9, 9E9, 9E9]];
    CONST robtarget p3561:= [[1444.5638364681504, 4.423399857044274, 993.500033578516], [0, 0, 1, 0], [0, 0, 0, 0], [9E9, 9E9, 9E9, 9E9, 9E9, 9E9]];
    CONST robtarget p3562:= [[1444.5945221601244, 4.750221146737246, 993.500033578516], [0, 0, 1, 0], [0, 0, 0, 0], [9E9, 9E9, 9E9, 9E9, 9E9, 9E9]];
    CONST robtarget p3563:= [[1444.6710804158372, 5.439612929627415, 993.500033578516], [0, 0, 1, 0], [0, 0, 0, 0], [9E9, 9E9, 9E9, 9E9, 9E9, 9E9]];
    CONST robtarget p3564:= [[1444.7059233943426, 5.756771017220018, 993.500033578516], [0, 0, 1, 0], [0, 0, 0, 0], [9E9, 9E9, 9E9, 9E9, 9E9, 9E9]];
    CONST robtarget p3565:= [[1444.7813864240288, 6.399868846253682, 993.500033578516], [0, 0, 1, 0], [0, 0, 0, 0], [9E9, 9E9, 9E9, 9E9, 9E9, 9E9]];
    CONST robtarget p3566:= [[1444.8621816645127, 7.0508629858633185, 993.500033578516], [0, 0, 1, 0], [0, 0, 0, 0], [9E9, 9E9, 9E9, 9E9, 9E9, 9E9]];
    CONST robtarget p3567:= [[1444.8862079695173, 7.395350083385225, 993.500033578516], [0, 0, 1, 0], [0, 0, 0, 0], [9E9, 9E9, 9E9, 9E9, 9E9, 9E9]];
    CONST robtarget p3568:= [[1444.9507516175283, 7.96420499306447, 993.500033578516], [0, 0, 1, 0], [0, 0, 0, 0], [9E9, 9E9, 9E9, 9E9, 9E9, 9E9]];
    CONST robtarget p3569:= [[1444.9643225395837, 8.06122200624199, 993.500033578516], [0, 0, 1, 0], [0, 0, 0, 0], [9E9, 9E9, 9E9, 9E9, 9E9, 9E9]];
    CONST robtarget p3570:= [[1445.006610153707, 8.340550046412304, 993.500033578516], [0, 0, 1, 0], [0, 0, 0, 0], [9E9, 9E9, 9E9, 9E9, 9E9, 9E9]];
    CONST robtarget p3571:= [[1445.1220891684259, 8.871981800045091, 993.500033578516], [0, 0, 1, 0], [0, 0, 0, 0], [9E9, 9E9, 9E9, 9E9, 9E9, 9E9]];
    CONST robtarget p3572:= [[1445.1453114117635, 9.006089570991321, 993.500033578516], [0, 0, 1, 0], [0, 0, 0, 0], [9E9, 9E9, 9E9, 9E9, 9E9, 9E9]];
    CONST robtarget p3573:= [[1445.2417461377509, 9.518825556421845, 993.500033578516], [0, 0, 1, 0], [0, 0, 0, 0], [9E9, 9E9, 9E9, 9E9, 9E9, 9E9]];
    CONST robtarget p3574:= [[1445.2680597934036, 9.721948112902098, 993.500033578516], [0, 0, 1, 0], [0, 0, 0, 0], [9E9, 9E9, 9E9, 9E9, 9E9, 9E9]];
    CONST robtarget p3575:= [[1445.2824501819928, 9.809116815332217, 993.500033578516], [0, 0, 1, 0], [0, 0, 0, 0], [9E9, 9E9, 9E9, 9E9, 9E9, 9E9]];
    CONST robtarget p3576:= [[1445.3158231956804, 9.985528260276467, 993.500033578516], [0, 0, 1, 0], [0, 0, 0, 0], [9E9, 9E9, 9E9, 9E9, 9E9, 9E9]];
    CONST robtarget p3577:= [[1445.4189728847298, 10.448378341408898, 993.500033578516], [0, 0, 1, 0], [0, 0, 0, 0], [9E9, 9E9, 9E9, 9E9, 9E9, 9E9]];
    CONST robtarget p3578:= [[1445.4737478292539, 10.73512926877379, 993.500033578516], [0, 0, 1, 0], [0, 0, 0, 0], [9E9, 9E9, 9E9, 9E9, 9E9, 9E9]];
    CONST robtarget p3579:= [[1445.5216283166671, 11.098489570658415, 993.500033578516], [0, 0, 1, 0], [0, 0, 0, 0], [9E9, 9E9, 9E9, 9E9, 9E9, 9E9]];
    CONST robtarget p3580:= [[1445.607844324445, 11.592914974054082, 993.500033578516], [0, 0, 1, 0], [0, 0, 0, 0], [9E9, 9E9, 9E9, 9E9, 9E9, 9E9]];
    CONST robtarget p3581:= [[1445.6465342912063, 11.782764377480092, 993.500033578516], [0, 0, 1, 0], [0, 0, 0, 0], [9E9, 9E9, 9E9, 9E9, 9E9, 9E9]];
    CONST robtarget p3582:= [[1445.6718525706506, 11.887893752436256, 993.500033578516], [0, 0, 1, 0], [0, 0, 0, 0], [9E9, 9E9, 9E9, 9E9, 9E9, 9E9]];
    CONST robtarget p3583:= [[1445.7335774426956, 12.182277578121344, 993.500033578516], [0, 0, 1, 0], [0, 0, 0, 0], [9E9, 9E9, 9E9, 9E9, 9E9, 9E9]];
    CONST robtarget p3584:= [[1445.7674247146101, 12.351660557892032, 993.500033578516], [0, 0, 1, 0], [0, 0, 0, 0], [9E9, 9E9, 9E9, 9E9, 9E9, 9E9]];
    CONST robtarget p3585:= [[1445.8384067939664, 12.60176605037536, 993.500033578516], [0, 0, 1, 0], [0, 0, 0, 0], [9E9, 9E9, 9E9, 9E9, 9E9, 9E9]];
    CONST robtarget p3586:= [[1445.9048383798565, 12.870160951727513, 993.500033578516], [0, 0, 1, 0], [0, 0, 0, 0], [9E9, 9E9, 9E9, 9E9, 9E9, 9E9]];
    CONST robtarget p3587:= [[1445.998214402726, 13.196687062136377, 993.500033578516], [0, 0, 1, 0], [0, 0, 0, 0], [9E9, 9E9, 9E9, 9E9, 9E9, 9E9]];
    CONST robtarget p3588:= [[1446.0463947546464, 13.402721705057857, 993.500033578516], [0, 0, 1, 0], [0, 0, 0, 0], [9E9, 9E9, 9E9, 9E9, 9E9, 9E9]];
    CONST robtarget p3589:= [[1446.1997438178155, 13.911869805080471, 993.500033578516], [0, 0, 1, 0], [0, 0, 0, 0], [9E9, 9E9, 9E9, 9E9, 9E9, 9E9]];
    CONST robtarget p3590:= [[1446.2762629473796, 14.245535715658704, 993.500033578516], [0, 0, 1, 0], [0, 0, 0, 0], [9E9, 9E9, 9E9, 9E9, 9E9, 9E9]];
    CONST robtarget p3591:= [[1446.3950136263534, 14.746056132894921, 993.500033578516], [0, 0, 1, 0], [0, 0, 0, 0], [9E9, 9E9, 9E9, 9E9, 9E9, 9E9]];
    CONST robtarget p3592:= [[1446.4997506124657, 15.08648877165038, 993.500033578516], [0, 0, 1, 0], [0, 0, 0, 0], [9E9, 9E9, 9E9, 9E9, 9E9, 9E9]];
    CONST robtarget p3593:= [[1446.575430012217, 15.404500244985172, 993.500033578516], [0, 0, 1, 0], [0, 0, 0, 0], [9E9, 9E9, 9E9, 9E9, 9E9, 9E9]];
    CONST robtarget p3594:= [[1446.6335092628235, 15.643524526965578, 993.500033578516], [0, 0, 1, 0], [0, 0, 0, 0], [9E9, 9E9, 9E9, 9E9, 9E9, 9E9]];
    CONST robtarget p3595:= [[1446.7031807526187, 15.890349156086373, 993.500033578516], [0, 0, 1, 0], [0, 0, 0, 0], [9E9, 9E9, 9E9, 9E9, 9E9, 9E9]];
    CONST robtarget p3596:= [[1446.749482642183, 16.077923135514027, 993.500033578516], [0, 0, 1, 0], [0, 0, 0, 0], [9E9, 9E9, 9E9, 9E9, 9E9, 9E9]];
    CONST robtarget p3597:= [[1446.8114590668554, 16.239465660020116, 993.500033578516], [0, 0, 1, 0], [0, 0, 0, 0], [9E9, 9E9, 9E9, 9E9, 9E9, 9E9]];
    CONST robtarget p3598:= [[1446.9146230357603, 16.53767565578663, 993.500033578516], [0, 0, 1, 0], [0, 0, 0, 0], [9E9, 9E9, 9E9, 9E9, 9E9, 9E9]];
    CONST robtarget p3599:= [[1446.963168670901, 16.66854774085074, 993.500033578516], [0, 0, 1, 0], [0, 0, 0, 0], [9E9, 9E9, 9E9, 9E9, 9E9, 9E9]];
    CONST robtarget p3600:= [[1446.9900299425199, 16.7425065795654, 993.500033578516], [0, 0, 1, 0], [0, 0, 0, 0], [9E9, 9E9, 9E9, 9E9, 9E9, 9E9]];
    CONST robtarget p3601:= [[1447.115491548474, 17.139664548150634, 993.500033578516], [0, 0, 1, 0], [0, 0, 0, 0], [9E9, 9E9, 9E9, 9E9, 9E9, 9E9]];
    CONST robtarget p3602:= [[1447.1389508457935, 17.22157378939157, 993.500033578516], [0, 0, 1, 0], [0, 0, 0, 0], [9E9, 9E9, 9E9, 9E9, 9E9, 9E9]];
    CONST robtarget p3603:= [[1447.291425586272, 17.63782814210286, 993.500033578516], [0, 0, 1, 0], [0, 0, 0, 0], [9E9, 9E9, 9E9, 9E9, 9E9, 9E9]];
    CONST robtarget p3604:= [[1447.3899407387735, 17.946634912413217, 993.500033578516], [0, 0, 1, 0], [0, 0, 0, 0], [9E9, 9E9, 9E9, 9E9, 9E9, 9E9]];
    CONST robtarget p3605:= [[1447.4383730731518, 18.098735357092124, 993.500033578516], [0, 0, 1, 0], [0, 0, 0, 0], [9E9, 9E9, 9E9, 9E9, 9E9, 9E9]];
    CONST robtarget p3606:= [[1447.565649674499, 18.435373736468506, 993.500033578516], [0, 0, 1, 0], [0, 0, 0, 0], [9E9, 9E9, 9E9, 9E9, 9E9, 9E9]];
    CONST robtarget p3607:= [[1447.6759540256755, 18.77435899441376, 993.500033578516], [0, 0, 1, 0], [0, 0, 0, 0], [9E9, 9E9, 9E9, 9E9, 9E9, 9E9]];
    CONST robtarget p3608:= [[1447.7180461341088, 18.8951522215865, 993.500033578516], [0, 0, 1, 0], [0, 0, 0, 0], [9E9, 9E9, 9E9, 9E9, 9E9, 9E9]];
    CONST robtarget p3609:= [[1447.9714600987909, 19.647451168715463, 993.500033578516], [0, 0, 1, 0], [0, 0, 0, 0], [9E9, 9E9, 9E9, 9E9, 9E9, 9E9]];
    CONST robtarget p3610:= [[1448.0516488997882, 19.887886445543487, 993.500033578516], [0, 0, 1, 0], [0, 0, 0, 0], [9E9, 9E9, 9E9, 9E9, 9E9, 9E9]];
    CONST robtarget p3611:= [[1448.0855779105252, 19.96749282121084, 993.500033578516], [0, 0, 1, 0], [0, 0, 0, 0], [9E9, 9E9, 9E9, 9E9, 9E9, 9E9]];
    CONST robtarget p3612:= [[1448.231774689219, 20.30060637761079, 993.500033578516], [0, 0, 1, 0], [0, 0, 0, 0], [9E9, 9E9, 9E9, 9E9, 9E9, 9E9]];
    CONST robtarget p3613:= [[1448.4249949476991, 20.771547217307756, 993.500033578516], [0, 0, 1, 0], [0, 0, 0, 0], [9E9, 9E9, 9E9, 9E9, 9E9, 9E9]];
    CONST robtarget p3614:= [[1448.4871546623035, 20.91339688820048, 993.500033578516], [0, 0, 1, 0], [0, 0, 0, 0], [9E9, 9E9, 9E9, 9E9, 9E9, 9E9]];
    CONST robtarget p3615:= [[1448.6708299281984, 21.346755088002624, 993.500033578516], [0, 0, 1, 0], [0, 0, 0, 0], [9E9, 9E9, 9E9, 9E9, 9E9, 9E9]];
    CONST robtarget p3616:= [[1448.9039866989838, 21.897020387037188, 993.500033578516], [0, 0, 1, 0], [0, 0, 0, 0], [9E9, 9E9, 9E9, 9E9, 9E9, 9E9]];
    CONST robtarget p3617:= [[1449.0517279863207, 22.251302004122692, 993.500033578516], [0, 0, 1, 0], [0, 0, 0, 0], [9E9, 9E9, 9E9, 9E9, 9E9, 9E9]];
    CONST robtarget p3618:= [[1449.2393358217416, 22.672920594804765, 993.500033578516], [0, 0, 1, 0], [0, 0, 0, 0], [9E9, 9E9, 9E9, 9E9, 9E9, 9E9]];
    CONST robtarget p3619:= [[1449.320061751566, 22.874129914388362, 993.500033578516], [0, 0, 1, 0], [0, 0, 0, 0], [9E9, 9E9, 9E9, 9E9, 9E9, 9E9]];
    CONST robtarget p3620:= [[1449.4529423222662, 23.175128115541014, 993.500033578516], [0, 0, 1, 0], [0, 0, 0, 0], [9E9, 9E9, 9E9, 9E9, 9E9, 9E9]];
    CONST robtarget p3621:= [[1449.4945941390156, 23.27668269252105, 993.500033578516], [0, 0, 1, 0], [0, 0, 0, 0], [9E9, 9E9, 9E9, 9E9, 9E9, 9E9]];
    CONST robtarget p3622:= [[1449.6231415702, 23.594832616201174, 993.500033578516], [0, 0, 1, 0], [0, 0, 0, 0], [9E9, 9E9, 9E9, 9E9, 9E9, 9E9]];
    CONST robtarget p3623:= [[1449.793827718006, 23.92004763440994, 993.500033578516], [0, 0, 1, 0], [0, 0, 0, 0], [9E9, 9E9, 9E9, 9E9, 9E9, 9E9]];
    CONST robtarget p3624:= [[1450.1388550638192, 24.583329948521325, 993.500033578516], [0, 0, 1, 0], [0, 0, 0, 0], [9E9, 9E9, 9E9, 9E9, 9E9, 9E9]];
    CONST robtarget p3625:= [[1450.2106914258848, 24.731601716591214, 993.500033578516], [0, 0, 1, 0], [0, 0, 0, 0], [9E9, 9E9, 9E9, 9E9, 9E9, 9E9]];
    CONST robtarget p3626:= [[1450.3869424847544, 25.078361949898607, 993.500033578516], [0, 0, 1, 0], [0, 0, 0, 0], [9E9, 9E9, 9E9, 9E9, 9E9, 9E9]];
    CONST robtarget p3627:= [[1450.4483093517806, 25.20364262778959, 993.500033578516], [0, 0, 1, 0], [0, 0, 0, 0], [9E9, 9E9, 9E9, 9E9, 9E9, 9E9]];
    CONST robtarget p3628:= [[1450.5592616233278, 25.41385635248946, 993.500033578516], [0, 0, 1, 0], [0, 0, 0, 0], [9E9, 9E9, 9E9, 9E9, 9E9, 9E9]];
    CONST robtarget p3629:= [[1450.6662676315955, 25.612184080744953, 993.500033578516], [0, 0, 1, 0], [0, 0, 0, 0], [9E9, 9E9, 9E9, 9E9, 9E9, 9E9]];
    CONST robtarget p3630:= [[1451.0725475657875, 26.41672561044352, 993.500033578516], [0, 0, 1, 0], [0, 0, 0, 0], [9E9, 9E9, 9E9, 9E9, 9E9, 9E9]];
    CONST robtarget p3631:= [[1451.452446368639, 27.11184788510795, 993.500033578516], [0, 0, 1, 0], [0, 0, 0, 0], [9E9, 9E9, 9E9, 9E9, 9E9, 9E9]];
    CONST robtarget p3632:= [[1451.5658213058541, 27.300875817009157, 993.500033578516], [0, 0, 1, 0], [0, 0, 0, 0], [9E9, 9E9, 9E9, 9E9, 9E9, 9E9]];
    CONST robtarget p3633:= [[1451.8239453307413, 27.775893752806056, 993.500033578516], [0, 0, 1, 0], [0, 0, 0, 0], [9E9, 9E9, 9E9, 9E9, 9E9, 9E9]];
    CONST robtarget p3634:= [[1451.8673058367597, 27.84268994217308, 993.500033578516], [0, 0, 1, 0], [0, 0, 0, 0], [9E9, 9E9, 9E9, 9E9, 9E9, 9E9]];
    CONST robtarget p3635:= [[1452.0289371690612, 28.094260015711797, 993.500033578516], [0, 0, 1, 0], [0, 0, 0, 0], [9E9, 9E9, 9E9, 9E9, 9E9, 9E9]];
    CONST robtarget p3636:= [[1452.207799621548, 28.38239021182298, 993.500033578516], [0, 0, 1, 0], [0, 0, 0, 0], [9E9, 9E9, 9E9, 9E9, 9E9, 9E9]];
    CONST robtarget p3637:= [[1452.2330896153153, 28.422617835947307, 993.500033578516], [0, 0, 1, 0], [0, 0, 0, 0], [9E9, 9E9, 9E9, 9E9, 9E9, 9E9]];
    CONST robtarget p3638:= [[1452.4619878307856, 28.792979689955587, 993.500033578516], [0, 0, 1, 0], [0, 0, 0, 0], [9E9, 9E9, 9E9, 9E9, 9E9, 9E9]];
    CONST robtarget p3639:= [[1452.533597025428, 28.905481381419136, 993.500033578516], [0, 0, 1, 0], [0, 0, 0, 0], [9E9, 9E9, 9E9, 9E9, 9E9, 9E9]];
    CONST robtarget p3640:= [[1452.8313620688805, 29.420512473147213, 993.500033578516], [0, 0, 1, 0], [0, 0, 0, 0], [9E9, 9E9, 9E9, 9E9, 9E9, 9E9]];
    CONST robtarget p3641:= [[1452.9340043735583, 29.58841246191679, 993.500033578516], [0, 0, 1, 0], [0, 0, 0, 0], [9E9, 9E9, 9E9, 9E9, 9E9, 9E9]];
    CONST robtarget p3642:= [[1453.0994544901425, 29.860442423281413, 993.500033578516], [0, 0, 1, 0], [0, 0, 0, 0], [9E9, 9E9, 9E9, 9E9, 9E9, 9E9]];
    CONST robtarget p3643:= [[1453.161528064843, 29.967482417793306, 993.500033578516], [0, 0, 1, 0], [0, 0, 0, 0], [9E9, 9E9, 9E9, 9E9, 9E9, 9E9]];
    CONST robtarget p3644:= [[1453.4513628373477, 30.44134602652609, 993.500033578516], [0, 0, 1, 0], [0, 0, 0, 0], [9E9, 9E9, 9E9, 9E9, 9E9, 9E9]];
    CONST robtarget p3645:= [[1453.6854707786879, 30.80483601238167, 993.500033578516], [0, 0, 1, 0], [0, 0, 0, 0], [9E9, 9E9, 9E9, 9E9, 9E9, 9E9]];
    CONST robtarget p3646:= [[1453.9211161267672, 31.114650239041666, 993.500033578516], [0, 0, 1, 0], [0, 0, 0, 0], [9E9, 9E9, 9E9, 9E9, 9E9, 9E9]];
    CONST robtarget p3647:= [[1454.1906046697188, 31.481268425394376, 993.500033578516], [0, 0, 1, 0], [0, 0, 0, 0], [9E9, 9E9, 9E9, 9E9, 9E9, 9E9]];
    CONST robtarget p3648:= [[1454.5510279769426, 32.0151606593429, 993.500033578516], [0, 0, 1, 0], [0, 0, 0, 0], [9E9, 9E9, 9E9, 9E9, 9E9, 9E9]];
    CONST robtarget p3649:= [[1454.7793086998495, 32.31517232566445, 993.500033578516], [0, 0, 1, 0], [0, 0, 0, 0], [9E9, 9E9, 9E9, 9E9, 9E9, 9E9]];
    CONST robtarget p3650:= [[1454.9334463041628, 32.534710785082495, 993.500033578516], [0, 0, 1, 0], [0, 0, 0, 0], [9E9, 9E9, 9E9, 9E9, 9E9, 9E9]];
    CONST robtarget p3651:= [[1455.1842969672346, 32.89992227249611, 993.500033578516], [0, 0, 1, 0], [0, 0, 0, 0], [9E9, 9E9, 9E9, 9E9, 9E9, 9E9]];
    CONST robtarget p3652:= [[1455.544377018847, 33.39548467522084, 993.500033578516], [0, 0, 1, 0], [0, 0, 0, 0], [9E9, 9E9, 9E9, 9E9, 9E9, 9E9]];
    CONST robtarget p3653:= [[1455.5897142851738, 33.452899994962095, 993.500033578516], [0, 0, 1, 0], [0, 0, 0, 0], [9E9, 9E9, 9E9, 9E9, 9E9, 9E9]];
    CONST robtarget p3654:= [[1455.9908168148902, 33.96803586779285, 993.500033578516], [0, 0, 1, 0], [0, 0, 0, 0], [9E9, 9E9, 9E9, 9E9, 9E9, 9E9]];
    CONST robtarget p3655:= [[1456.142873917458, 34.177226410628265, 993.500033578516], [0, 0, 1, 0], [0, 0, 0, 0], [9E9, 9E9, 9E9, 9E9, 9E9, 9E9]];
    CONST robtarget p3656:= [[1456.2861120950479, 34.37132553025879, 993.500033578516], [0, 0, 1, 0], [0, 0, 0, 0], [9E9, 9E9, 9E9, 9E9, 9E9, 9E9]];
    CONST robtarget p3657:= [[1456.3808671941704, 34.489732802273934, 993.500033578516], [0, 0, 1, 0], [0, 0, 0, 0], [9E9, 9E9, 9E9, 9E9, 9E9, 9E9]];
    CONST robtarget p3658:= [[1456.5183956713365, 34.6508578040569, 993.500033578516], [0, 0, 1, 0], [0, 0, 0, 0], [9E9, 9E9, 9E9, 9E9, 9E9, 9E9]];
    CONST robtarget p3659:= [[1456.5648954310695, 34.701588905945684, 993.500033578516], [0, 0, 1, 0], [0, 0, 0, 0], [9E9, 9E9, 9E9, 9E9, 9E9, 9E9]];
    CONST robtarget p3660:= [[1456.9926046570513, 35.20351088932067, 993.500033578516], [0, 0, 1, 0], [0, 0, 0, 0], [9E9, 9E9, 9E9, 9E9, 9E9, 9E9]];
    CONST robtarget p3661:= [[1457.24496154393, 35.51563986935939, 993.500033578516], [0, 0, 1, 0], [0, 0, 0, 0], [9E9, 9E9, 9E9, 9E9, 9E9, 9E9]];
    CONST robtarget p3662:= [[1457.3841303580239, 35.698471375179096, 993.500033578516], [0, 0, 1, 0], [0, 0, 0, 0], [9E9, 9E9, 9E9, 9E9, 9E9, 9E9]];
    CONST robtarget p3663:= [[1457.7753380052272, 36.16347899292073, 993.500033578516], [0, 0, 1, 0], [0, 0, 0, 0], [9E9, 9E9, 9E9, 9E9, 9E9, 9E9]];
    CONST robtarget p3664:= [[1457.8825686691912, 36.29821057724298, 993.500033578516], [0, 0, 1, 0], [0, 0, 0, 0], [9E9, 9E9, 9E9, 9E9, 9E9, 9E9]];
    CONST robtarget p3665:= [[1457.9288417125629, 36.350461248352104, 993.500033578516], [0, 0, 1, 0], [0, 0, 0, 0], [9E9, 9E9, 9E9, 9E9, 9E9, 9E9]];
    CONST robtarget p3666:= [[1458.325343420478, 36.830194950615535, 993.500033578516], [0, 0, 1, 0], [0, 0, 0, 0], [9E9, 9E9, 9E9, 9E9, 9E9, 9E9]];
    CONST robtarget p3667:= [[1458.5644231500794, 37.105481478684325, 993.500033578516], [0, 0, 1, 0], [0, 0, 0, 0], [9E9, 9E9, 9E9, 9E9, 9E9, 9E9]];
    CONST robtarget p3668:= [[1458.657161763589, 37.20545661712026, 993.500033578516], [0, 0, 1, 0], [0, 0, 0, 0], [9E9, 9E9, 9E9, 9E9, 9E9, 9E9]];
    CONST robtarget p3669:= [[1459.003490955316, 37.554222315940905, 993.500033578516], [0, 0, 1, 0], [0, 0, 0, 0], [9E9, 9E9, 9E9, 9E9, 9E9, 9E9]];
    CONST robtarget p3670:= [[1459.4011270455276, 37.959443622489516, 993.500033578516], [0, 0, 1, 0], [0, 0, 0, 0], [9E9, 9E9, 9E9, 9E9, 9E9, 9E9]];
    CONST robtarget p3671:= [[1459.46914321446, 38.0360744832296, 993.500033578516], [0, 0, 1, 0], [0, 0, 0, 0], [9E9, 9E9, 9E9, 9E9, 9E9, 9E9]];
    CONST robtarget p3672:= [[1459.8749096630363, 38.47245950838625, 993.500033578516], [0, 0, 1, 0], [0, 0, 0, 0], [9E9, 9E9, 9E9, 9E9, 9E9, 9E9]];
    CONST robtarget p3673:= [[1459.9588148801308, 38.556081048127666, 993.500033578516], [0, 0, 1, 0], [0, 0, 0, 0], [9E9, 9E9, 9E9, 9E9, 9E9, 9E9]];
    CONST robtarget p3674:= [[1460.3510310184624, 38.96185371932967, 993.500033578516], [0, 0, 1, 0], [0, 0, 0, 0], [9E9, 9E9, 9E9, 9E9, 9E9, 9E9]];
    CONST robtarget p3675:= [[1460.617130121585, 39.23007269322247, 993.500033578516], [0, 0, 1, 0], [0, 0, 0, 0], [9E9, 9E9, 9E9, 9E9, 9E9, 9E9]];
    CONST robtarget p3676:= [[1460.8576757027458, 39.479066375882866, 993.500033578516], [0, 0, 1, 0], [0, 0, 0, 0], [9E9, 9E9, 9E9, 9E9, 9E9, 9E9]];
    CONST robtarget p3677:= [[1460.99945380179, 39.62918694839891, 993.500033578516], [0, 0, 1, 0], [0, 0, 0, 0], [9E9, 9E9, 9E9, 9E9, 9E9, 9E9]];
    CONST robtarget p3678:= [[1461.3831763263606, 40.039883492308775, 993.500033578516], [0, 0, 1, 0], [0, 0, 0, 0], [9E9, 9E9, 9E9, 9E9, 9E9, 9E9]];
    CONST robtarget p3679:= [[1461.663956978733, 40.2841403366988, 993.500033578516], [0, 0, 1, 0], [0, 0, 0, 0], [9E9, 9E9, 9E9, 9E9, 9E9, 9E9]];
    CONST robtarget p3680:= [[1461.757610135975, 40.3723412493019, 993.500033578516], [0, 0, 1, 0], [0, 0, 0, 0], [9E9, 9E9, 9E9, 9E9, 9E9, 9E9]];
    CONST robtarget p3681:= [[1462.0725048199401, 40.64224046388573, 993.500033578516], [0, 0, 1, 0], [0, 0, 0, 0], [9E9, 9E9, 9E9, 9E9, 9E9, 9E9]];
    CONST robtarget p3682:= [[1462.3445196139703, 40.89199147939398, 993.500033578516], [0, 0, 1, 0], [0, 0, 0, 0], [9E9, 9E9, 9E9, 9E9, 9E9, 9E9]];
    CONST robtarget p3683:= [[1462.561492598222, 41.076753381821206, 993.500033578516], [0, 0, 1, 0], [0, 0, 0, 0], [9E9, 9E9, 9E9, 9E9, 9E9, 9E9]];
    CONST robtarget p3684:= [[1462.6594978099988, 41.16310651974423, 993.500033578516], [0, 0, 1, 0], [0, 0, 0, 0], [9E9, 9E9, 9E9, 9E9, 9E9, 9E9]];
    CONST robtarget p3685:= [[1462.9750698440216, 41.465493397367425, 993.500033578516], [0, 0, 1, 0], [0, 0, 0, 0], [9E9, 9E9, 9E9, 9E9, 9E9, 9E9]];
    CONST robtarget p3686:= [[1463.062540648459, 41.5438304429655, 993.500033578516], [0, 0, 1, 0], [0, 0, 0, 0], [9E9, 9E9, 9E9, 9E9, 9E9, 9E9]];
    CONST robtarget p3687:= [[1463.3039194311914, 41.75740415497293, 993.500033578516], [0, 0, 1, 0], [0, 0, 0, 0], [9E9, 9E9, 9E9, 9E9, 9E9, 9E9]];
    CONST robtarget p3688:= [[1463.683506573706, 42.09837138506629, 993.500033578516], [0, 0, 1, 0], [0, 0, 0, 0], [9E9, 9E9, 9E9, 9E9, 9E9, 9E9]];
    CONST robtarget p3689:= [[1464.0250487506437, 42.40696731839559, 993.500033578516], [0, 0, 1, 0], [0, 0, 0, 0], [9E9, 9E9, 9E9, 9E9, 9E9, 9E9]];
    CONST robtarget p3690:= [[1464.3929686746292, 42.73661176112732, 993.500033578516], [0, 0, 1, 0], [0, 0, 0, 0], [9E9, 9E9, 9E9, 9E9, 9E9, 9E9]];
    CONST robtarget p3691:= [[1464.539737174689, 42.83932740418268, 993.500033578516], [0, 0, 1, 0], [0, 0, 0, 0], [9E9, 9E9, 9E9, 9E9, 9E9, 9E9]];
    CONST robtarget p3692:= [[1464.7592769986597, 43.00621666861372, 993.500033578516], [0, 0, 1, 0], [0, 0, 0, 0], [9E9, 9E9, 9E9, 9E9, 9E9, 9E9]];
    CONST robtarget p3693:= [[1464.779244173724, 43.02055174407589, 993.500033578516], [0, 0, 1, 0], [0, 0, 0, 0], [9E9, 9E9, 9E9, 9E9, 9E9, 9E9]];
    CONST robtarget p3694:= [[1465.2344931411096, 43.35290425777251, 993.500033578516], [0, 0, 1, 0], [0, 0, 0, 0], [9E9, 9E9, 9E9, 9E9, 9E9, 9E9]];
    CONST robtarget p3695:= [[1465.4867172775403, 43.57422668485684, 993.500033578516], [0, 0, 1, 0], [0, 0, 0, 0], [9E9, 9E9, 9E9, 9E9, 9E9, 9E9]];
    CONST robtarget p3696:= [[1465.8537483773935, 43.849589256079355, 993.500033578516], [0, 0, 1, 0], [0, 0, 0, 0], [9E9, 9E9, 9E9, 9E9, 9E9, 9E9]];
    CONST robtarget p3697:= [[1466.170681513625, 44.079449669616096, 993.500033578516], [0, 0, 1, 0], [0, 0, 0, 0], [9E9, 9E9, 9E9, 9E9, 9E9, 9E9]];
    CONST robtarget p3698:= [[1466.6684553085745, 44.4839922033228, 993.500033578516], [0, 0, 1, 0], [0, 0, 0, 0], [9E9, 9E9, 9E9, 9E9, 9E9, 9E9]];
    CONST robtarget p3699:= [[1466.908595941648, 44.66628747791145, 993.500033578516], [0, 0, 1, 0], [0, 0, 0, 0], [9E9, 9E9, 9E9, 9E9, 9E9, 9E9]];
    CONST robtarget p3700:= [[1467.4085555099596, 45.06247014559955, 993.500033578516], [0, 0, 1, 0], [0, 0, 0, 0], [9E9, 9E9, 9E9, 9E9, 9E9, 9E9]];
    CONST robtarget p3701:= [[1467.5901955496547, 45.198671673614854, 993.500033578516], [0, 0, 1, 0], [0, 0, 0, 0], [9E9, 9E9, 9E9, 9E9, 9E9, 9E9]];
    CONST robtarget p3702:= [[1467.9821576986867, 45.455434248663735, 993.500033578516], [0, 0, 1, 0], [0, 0, 0, 0], [9E9, 9E9, 9E9, 9E9, 9E9, 9E9]];
    CONST robtarget p3703:= [[1468.1803314044782, 45.592242616822716, 993.500033578516], [0, 0, 1, 0], [0, 0, 0, 0], [9E9, 9E9, 9E9, 9E9, 9E9, 9E9]];
    CONST robtarget p3704:= [[1468.3733053958097, 45.72519930377871, 993.500033578516], [0, 0, 1, 0], [0, 0, 0, 0], [9E9, 9E9, 9E9, 9E9, 9E9, 9E9]];
    CONST robtarget p3705:= [[1468.7273978480455, 45.94679084755978, 993.500033578516], [0, 0, 1, 0], [0, 0, 0, 0], [9E9, 9E9, 9E9, 9E9, 9E9, 9E9]];
    CONST robtarget p3706:= [[1469.2168845064773, 46.254115153217185, 993.500033578516], [0, 0, 1, 0], [0, 0, 0, 0], [9E9, 9E9, 9E9, 9E9, 9E9, 9E9]];
    CONST robtarget p3707:= [[1469.526544359998, 46.471423673989634, 993.500033578516], [0, 0, 1, 0], [0, 0, 0, 0], [9E9, 9E9, 9E9, 9E9, 9E9, 9E9]];
    CONST robtarget p3708:= [[1469.8544449572703, 46.71200469707887, 993.500033578516], [0, 0, 1, 0], [0, 0, 0, 0], [9E9, 9E9, 9E9, 9E9, 9E9, 9E9]];
    CONST robtarget p3709:= [[1470.1511702040896, 46.90230613321492, 993.500033578516], [0, 0, 1, 0], [0, 0, 0, 0], [9E9, 9E9, 9E9, 9E9, 9E9, 9E9]];
    CONST robtarget p3710:= [[1470.5790929705583, 47.17604478326052, 993.500033578516], [0, 0, 1, 0], [0, 0, 0, 0], [9E9, 9E9, 9E9, 9E9, 9E9, 9E9]];
    CONST robtarget p3711:= [[1470.7730334383841, 47.29359744333901, 993.500033578516], [0, 0, 1, 0], [0, 0, 0, 0], [9E9, 9E9, 9E9, 9E9, 9E9, 9E9]];
    CONST robtarget p3712:= [[1471.138211878014, 47.54256963900757, 993.500033578516], [0, 0, 1, 0], [0, 0, 0, 0], [9E9, 9E9, 9E9, 9E9, 9E9, 9E9]];
    CONST robtarget p3713:= [[1471.2995140543833, 47.63608204772923, 993.500033578516], [0, 0, 1, 0], [0, 0, 0, 0], [9E9, 9E9, 9E9, 9E9, 9E9, 9E9]];
    CONST robtarget p3714:= [[1471.705834503272, 47.86692071630604, 993.500033578516], [0, 0, 1, 0], [0, 0, 0, 0], [9E9, 9E9, 9E9, 9E9, 9E9, 9E9]];
    CONST robtarget p3715:= [[1472.2583850180765, 48.17188903678078, 993.500033578516], [0, 0, 1, 0], [0, 0, 0, 0], [9E9, 9E9, 9E9, 9E9, 9E9, 9E9]];
    CONST robtarget p3716:= [[1472.5432201664291, 48.31772617751973, 993.500033578516], [0, 0, 1, 0], [0, 0, 0, 0], [9E9, 9E9, 9E9, 9E9, 9E9, 9E9]];
    CONST robtarget p3717:= [[1473.154705121749, 48.6785785389972, 993.500033578516], [0, 0, 1, 0], [0, 0, 0, 0], [9E9, 9E9, 9E9, 9E9, 9E9, 9E9]];
    CONST robtarget p3718:= [[1473.8577735180359, 49.07163965929648, 993.500033578516], [0, 0, 1, 0], [0, 0, 0, 0], [9E9, 9E9, 9E9, 9E9, 9E9, 9E9]];
    CONST robtarget p3719:= [[1474.2407937417188, 49.28997948578946, 993.500033578516], [0, 0, 1, 0], [0, 0, 0, 0], [9E9, 9E9, 9E9, 9E9, 9E9, 9E9]];
    CONST robtarget p3720:= [[1474.459403458237, 49.40910658903098, 993.500033578516], [0, 0, 1, 0], [0, 0, 0, 0], [9E9, 9E9, 9E9, 9E9, 9E9, 9E9]];
    CONST robtarget p3721:= [[1474.7442864938873, 49.55154892245446, 993.500033578516], [0, 0, 1, 0], [0, 0, 0, 0], [9E9, 9E9, 9E9, 9E9, 9E9, 9E9]];
    CONST robtarget p3722:= [[1475.0354078606038, 49.685378032135446, 993.500033578516], [0, 0, 1, 0], [0, 0, 0, 0], [9E9, 9E9, 9E9, 9E9, 9E9, 9E9]];
    CONST robtarget p3723:= [[1475.226908783592, 49.77365218761719, 993.500033578516], [0, 0, 1, 0], [0, 0, 0, 0], [9E9, 9E9, 9E9, 9E9, 9E9, 9E9]];
    CONST robtarget p3724:= [[1475.5441998671356, 49.92405775651065, 993.500033578516], [0, 0, 1, 0], [0, 0, 0, 0], [9E9, 9E9, 9E9, 9E9, 9E9, 9E9]];
    CONST robtarget p3725:= [[1475.6972422036588, 49.99986216350625, 993.500033578516], [0, 0, 1, 0], [0, 0, 0, 0], [9E9, 9E9, 9E9, 9E9, 9E9, 9E9]];
    CONST robtarget p3726:= [[1476.440655056434, 50.34763191632996, 993.500033578516], [0, 0, 1, 0], [0, 0, 0, 0], [9E9, 9E9, 9E9, 9E9, 9E9, 9E9]];
    CONST robtarget p3727:= [[1476.4890589479348, 50.373203547174995, 993.500033578516], [0, 0, 1, 0], [0, 0, 0, 0], [9E9, 9E9, 9E9, 9E9, 9E9, 9E9]];
    CONST robtarget p3728:= [[1476.7531433229328, 50.49628331428126, 993.500033578516], [0, 0, 1, 0], [0, 0, 0, 0], [9E9, 9E9, 9E9, 9E9, 9E9, 9E9]];
    CONST robtarget p3729:= [[1476.949853517882, 50.58505586005572, 993.500033578516], [0, 0, 1, 0], [0, 0, 0, 0], [9E9, 9E9, 9E9, 9E9, 9E9, 9E9]];
    CONST robtarget p3730:= [[1477.4658084417183, 50.82128179312423, 993.500033578516], [0, 0, 1, 0], [0, 0, 0, 0], [9E9, 9E9, 9E9, 9E9, 9E9, 9E9]];
    CONST robtarget p3731:= [[1477.5788960110544, 50.87934957316452, 993.500033578516], [0, 0, 1, 0], [0, 0, 0, 0], [9E9, 9E9, 9E9, 9E9, 9E9, 9E9]];
    CONST robtarget p3732:= [[1477.9542911050394, 51.060875359104855, 993.500033578516], [0, 0, 1, 0], [0, 0, 0, 0], [9E9, 9E9, 9E9, 9E9, 9E9, 9E9]];
    CONST robtarget p3733:= [[1478.1978333252403, 51.15743577038779, 993.500033578516], [0, 0, 1, 0], [0, 0, 0, 0], [9E9, 9E9, 9E9, 9E9, 9E9, 9E9]];
    CONST robtarget p3734:= [[1478.536090108392, 51.29448411684767, 993.500033578516], [0, 0, 1, 0], [0, 0, 0, 0], [9E9, 9E9, 9E9, 9E9, 9E9, 9E9]];
    CONST robtarget p3735:= [[1478.704665605398, 51.36738007568766, 993.500033578516], [0, 0, 1, 0], [0, 0, 0, 0], [9E9, 9E9, 9E9, 9E9, 9E9, 9E9]];
    CONST robtarget p3736:= [[1478.9490499141973, 51.46205148022503, 993.500033578516], [0, 0, 1, 0], [0, 0, 0, 0], [9E9, 9E9, 9E9, 9E9, 9E9, 9E9]];
    CONST robtarget p3737:= [[1479.2201069572473, 51.55212740909984, 993.500033578516], [0, 0, 1, 0], [0, 0, 0, 0], [9E9, 9E9, 9E9, 9E9, 9E9, 9E9]];
    CONST robtarget p3738:= [[1479.4093772257177, 51.62254437359674, 993.500033578516], [0, 0, 1, 0], [0, 0, 0, 0], [9E9, 9E9, 9E9, 9E9, 9E9, 9E9]];
    CONST robtarget p3739:= [[1479.884107863292, 51.82290066118131, 993.500033578516], [0, 0, 1, 0], [0, 0, 0, 0], [9E9, 9E9, 9E9, 9E9, 9E9, 9E9]];
    CONST robtarget p3740:= [[1480.0219738860078, 51.87390745635038, 993.500033578516], [0, 0, 1, 0], [0, 0, 0, 0], [9E9, 9E9, 9E9, 9E9, 9E9, 9E9]];
    CONST robtarget p3741:= [[1480.3122672382174, 51.97516831926167, 993.500033578516], [0, 0, 1, 0], [0, 0, 0, 0], [9E9, 9E9, 9E9, 9E9, 9E9, 9E9]];
    CONST robtarget p3742:= [[1480.5127659170769, 52.052599503248516, 993.500033578516], [0, 0, 1, 0], [0, 0, 0, 0], [9E9, 9E9, 9E9, 9E9, 9E9, 9E9]];
    CONST robtarget p3743:= [[1480.9527504718317, 52.21887897185981, 993.500033578516], [0, 0, 1, 0], [0, 0, 0, 0], [9E9, 9E9, 9E9, 9E9, 9E9, 9E9]];
    CONST robtarget p3744:= [[1480.9975336909815, 52.23409006883709, 993.500033578516], [0, 0, 1, 0], [0, 0, 0, 0], [9E9, 9E9, 9E9, 9E9, 9E9, 9E9]];
    CONST robtarget p3745:= [[1481.6525885806861, 52.49640372020842, 993.500033578516], [0, 0, 1, 0], [0, 0, 0, 0], [9E9, 9E9, 9E9, 9E9, 9E9, 9E9]];
    CONST robtarget p3746:= [[1482.1722562199236, 52.67859573487799, 993.500033578516], [0, 0, 1, 0], [0, 0, 0, 0], [9E9, 9E9, 9E9, 9E9, 9E9, 9E9]];
    CONST robtarget p3747:= [[1482.422468498166, 52.75255705558391, 993.500033578516], [0, 0, 1, 0], [0, 0, 0, 0], [9E9, 9E9, 9E9, 9E9, 9E9, 9E9]];
    CONST robtarget p3748:= [[1482.7591760605947, 52.85444690126853, 993.500033578516], [0, 0, 1, 0], [0, 0, 0, 0], [9E9, 9E9, 9E9, 9E9, 9E9, 9E9]];
    CONST robtarget p3749:= [[1482.950187226955, 52.9101844568785, 993.500033578516], [0, 0, 1, 0], [0, 0, 0, 0], [9E9, 9E9, 9E9, 9E9, 9E9, 9E9]];
    CONST robtarget p3750:= [[1483.8544949333061, 53.18390796207564, 993.500033578516], [0, 0, 1, 0], [0, 0, 0, 0], [9E9, 9E9, 9E9, 9E9, 9E9, 9E9]];
    CONST robtarget p3751:= [[1484.2936015321861, 53.3009952773625, 993.500033578516], [0, 0, 1, 0], [0, 0, 0, 0], [9E9, 9E9, 9E9, 9E9, 9E9, 9E9]];
    CONST robtarget p3752:= [[1484.5174562432728, 53.36557938648234, 993.500033578516], [0, 0, 1, 0], [0, 0, 0, 0], [9E9, 9E9, 9E9, 9E9, 9E9, 9E9]];
    CONST robtarget p3753:= [[1484.7326020812595, 53.436117344545025, 993.500033578516], [0, 0, 1, 0], [0, 0, 0, 0], [9E9, 9E9, 9E9, 9E9, 9E9, 9E9]];
    CONST robtarget p3754:= [[1484.8983132290791, 53.4779007467376, 993.500033578516], [0, 0, 1, 0], [0, 0, 0, 0], [9E9, 9E9, 9E9, 9E9, 9E9, 9E9]];
    CONST robtarget p3755:= [[1485.5216835316946, 53.67750934703089, 993.500033578516], [0, 0, 1, 0], [0, 0, 0, 0], [9E9, 9E9, 9E9, 9E9, 9E9, 9E9]];
    CONST robtarget p3756:= [[1485.7477022406886, 53.75038732419226, 993.500033578516], [0, 0, 1, 0], [0, 0, 0, 0], [9E9, 9E9, 9E9, 9E9, 9E9, 9E9]];
    CONST robtarget p3757:= [[1485.9218122449201, 53.802657113074204, 993.500033578516], [0, 0, 1, 0], [0, 0, 0, 0], [9E9, 9E9, 9E9, 9E9, 9E9, 9E9]];
    CONST robtarget p3758:= [[1486.0749817177636, 53.83536129152114, 993.500033578516], [0, 0, 1, 0], [0, 0, 0, 0], [9E9, 9E9, 9E9, 9E9, 9E9, 9E9]];
    CONST robtarget p3759:= [[1486.4207648037536, 53.92356836520794, 993.500033578516], [0, 0, 1, 0], [0, 0, 0, 0], [9E9, 9E9, 9E9, 9E9, 9E9, 9E9]];
    CONST robtarget p3760:= [[1486.4671398670203, 53.93180005249839, 993.500033578516], [0, 0, 1, 0], [0, 0, 0, 0], [9E9, 9E9, 9E9, 9E9, 9E9, 9E9]];
    CONST robtarget p3761:= [[1486.6446076759983, 53.965180547458814, 993.500033578516], [0, 0, 1, 0], [0, 0, 0, 0], [9E9, 9E9, 9E9, 9E9, 9E9, 9E9]];
    CONST robtarget p3762:= [[1486.9064600720542, 54.0258102375126, 993.500033578516], [0, 0, 1, 0], [0, 0, 0, 0], [9E9, 9E9, 9E9, 9E9, 9E9, 9E9]];
    CONST robtarget p3763:= [[1487.0232288487753, 54.05740655329794, 993.500033578516], [0, 0, 1, 0], [0, 0, 0, 0], [9E9, 9E9, 9E9, 9E9, 9E9, 9E9]];
    CONST robtarget p3764:= [[1487.2504485114237, 54.110056444868746, 993.500033578516], [0, 0, 1, 0], [0, 0, 0, 0], [9E9, 9E9, 9E9, 9E9, 9E9, 9E9]];
    CONST robtarget p3765:= [[1487.9308386438315, 54.2560729637226, 993.500033578516], [0, 0, 1, 0], [0, 0, 0, 0], [9E9, 9E9, 9E9, 9E9, 9E9, 9E9]];
    CONST robtarget p3766:= [[1488.0284733352564, 54.28476002764231, 993.500033578516], [0, 0, 1, 0], [0, 0, 0, 0], [9E9, 9E9, 9E9, 9E9, 9E9, 9E9]];
    CONST robtarget p3767:= [[1488.2091107772355, 54.323471223132586, 993.500033578516], [0, 0, 1, 0], [0, 0, 0, 0], [9E9, 9E9, 9E9, 9E9, 9E9, 9E9]];
    CONST robtarget p3768:= [[1488.892618827427, 54.47604600326335, 993.500033578516], [0, 0, 1, 0], [0, 0, 0, 0], [9E9, 9E9, 9E9, 9E9, 9E9, 9E9]];
    CONST robtarget p3769:= [[1489.204454295672, 54.53617576679217, 993.500033578516], [0, 0, 1, 0], [0, 0, 0, 0], [9E9, 9E9, 9E9, 9E9, 9E9, 9E9]];
    CONST robtarget p3770:= [[1489.6050625910536, 54.62900538338101, 993.500033578516], [0, 0, 1, 0], [0, 0, 0, 0], [9E9, 9E9, 9E9, 9E9, 9E9, 9E9]];
    CONST robtarget p3771:= [[1490.050690375515, 54.70607212148511, 993.500033578516], [0, 0, 1, 0], [0, 0, 0, 0], [9E9, 9E9, 9E9, 9E9, 9E9, 9E9]];
    CONST robtarget p3772:= [[1490.1143241236448, 54.71922648721541, 993.500033578516], [0, 0, 1, 0], [0, 0, 0, 0], [9E9, 9E9, 9E9, 9E9, 9E9, 9E9]];
    CONST robtarget p3773:= [[1490.237705262652, 54.739315243549584, 993.500033578516], [0, 0, 1, 0], [0, 0, 0, 0], [9E9, 9E9, 9E9, 9E9, 9E9, 9E9]];
    CONST robtarget p3774:= [[1490.990526638497, 54.85844121346756, 993.500033578516], [0, 0, 1, 0], [0, 0, 0, 0], [9E9, 9E9, 9E9, 9E9, 9E9, 9E9]];
    CONST robtarget p3775:= [[1491.4624165374887, 54.92594792625802, 993.500033578516], [0, 0, 1, 0], [0, 0, 0, 0], [9E9, 9E9, 9E9, 9E9, 9E9, 9E9]];
    CONST robtarget p3776:= [[1491.7342812721936, 54.95632817058069, 993.500033578516], [0, 0, 1, 0], [0, 0, 0, 0], [9E9, 9E9, 9E9, 9E9, 9E9, 9E9]];
    CONST robtarget p3777:= [[1492.4129038485682, 55.05878992085222, 993.500033578516], [0, 0, 1, 0], [0, 0, 0, 0], [9E9, 9E9, 9E9, 9E9, 9E9, 9E9]];
    CONST robtarget p3778:= [[1492.9380760741176, 55.142570966788256, 993.500033578516], [0, 0, 1, 0], [0, 0, 0, 0], [9E9, 9E9, 9E9, 9E9, 9E9, 9E9]];
    CONST robtarget p3779:= [[1493.6941482147506, 55.24893674094237, 993.500033578516], [0, 0, 1, 0], [0, 0, 0, 0], [9E9, 9E9, 9E9, 9E9, 9E9, 9E9]];
    CONST robtarget p3780:= [[1494.0158957346061, 55.298830300586616, 993.500033578516], [0, 0, 1, 0], [0, 0, 0, 0], [9E9, 9E9, 9E9, 9E9, 9E9, 9E9]];
    CONST robtarget p3781:= [[1494.3761904222424, 55.32510949564299, 993.500033578516], [0, 0, 1, 0], [0, 0, 0, 0], [9E9, 9E9, 9E9, 9E9, 9E9, 9E9]];
    CONST robtarget p3782:= [[1494.543298392665, 55.33230802274724, 993.500033578516], [0, 0, 1, 0], [0, 0, 0, 0], [9E9, 9E9, 9E9, 9E9, 9E9, 9E9]];
    CONST robtarget p3783:= [[1494.7354423666843, 55.347120782798385, 993.500033578516], [0, 0, 1, 0], [0, 0, 0, 0], [9E9, 9E9, 9E9, 9E9, 9E9, 9E9]];
    CONST robtarget p3784:= [[1495.2507916550298, 55.38738263579718, 993.500033578516], [0, 0, 1, 0], [0, 0, 0, 0], [9E9, 9E9, 9E9, 9E9, 9E9, 9E9]];
    CONST robtarget p3785:= [[1496.072581611918, 55.44347519649516, 993.500033578516], [0, 0, 1, 0], [0, 0, 0, 0], [9E9, 9E9, 9E9, 9E9, 9E9, 9E9]];
    CONST robtarget p3786:= [[1496.2822980375445, 55.461064449626264, 993.500033578516], [0, 0, 1, 0], [0, 0, 0, 0], [9E9, 9E9, 9E9, 9E9, 9E9, 9E9]];
    CONST robtarget p3787:= [[1496.3469431294936, 55.46401629013933, 993.500033578516], [0, 0, 1, 0], [0, 0, 0, 0], [9E9, 9E9, 9E9, 9E9, 9E9, 9E9]];
    CONST robtarget p3788:= [[1496.7949346567718, 55.49194629748945, 993.500033578516], [0, 0, 1, 0], [0, 0, 0, 0], [9E9, 9E9, 9E9, 9E9, 9E9, 9E9]];
    CONST robtarget p3789:= [[1496.9326025885246, 55.495649153389465, 993.500033578516], [0, 0, 1, 0], [0, 0, 0, 0], [9E9, 9E9, 9E9, 9E9, 9E9, 9E9]];
    CONST robtarget p3790:= [[1497.0763530974082, 55.503204063764485, 993.500033578516], [0, 0, 1, 0], [0, 0, 0, 0], [9E9, 9E9, 9E9, 9E9, 9E9, 9E9]];
    CONST robtarget p3791:= [[1497.5233000040034, 55.52784080655721, 993.500033578516], [0, 0, 1, 0], [0, 0, 0, 0], [9E9, 9E9, 9E9, 9E9, 9E9, 9E9]];
    CONST robtarget p3792:= [[1497.7915736446887, 55.56086512210264, 993.500033578516], [0, 0, 1, 0], [0, 0, 0, 0], [9E9, 9E9, 9E9, 9E9, 9E9, 9E9]];
    CONST robtarget p3793:= [[1497.9848881977885, 55.585857485792445, 993.500033578516], [0, 0, 1, 0], [0, 0, 0, 0], [9E9, 9E9, 9E9, 9E9, 9E9, 9E9]];
    CONST robtarget p3794:= [[1498.3477380520449, 55.56868397836483, 993.500033578516], [0, 0, 1, 0], [0, 0, 0, 0], [9E9, 9E9, 9E9, 9E9, 9E9, 9E9]];
    CONST robtarget p3795:= [[1498.9099574409727, 55.57686311057218, 993.500033578516], [0, 0, 1, 0], [0, 0, 0, 0], [9E9, 9E9, 9E9, 9E9, 9E9, 9E9]];
    CONST robtarget p3796:= [[1499.22659845426, 55.58202077521706, 993.500033578516], [0, 0, 1, 0], [0, 0, 0, 0], [9E9, 9E9, 9E9, 9E9, 9E9, 9E9]];
    CONST robtarget p3797:= [[1499.6370770124408, 55.57998779262671, 993.500033578516], [0, 0, 1, 0], [0, 0, 0, 0], [9E9, 9E9, 9E9, 9E9, 9E9, 9E9]];
    CONST robtarget p3798:= [[1499.7905785939129, 55.577307717627434, 993.500033578516], [0, 0, 1, 0], [0, 0, 0, 0], [9E9, 9E9, 9E9, 9E9, 9E9, 9E9]];
    CONST robtarget p3799:= [[1499.888226279698, 55.574475834083344, 993.500033578516], [0, 0, 1, 0], [0, 0, 0, 0], [9E9, 9E9, 9E9, 9E9, 9E9, 9E9]];
    CONST robtarget p3800:= [[1500.400207165641, 55.584447974632866, 993.500033578516], [0, 0, 1, 0], [0, 0, 0, 0], [9E9, 9E9, 9E9, 9E9, 9E9, 9E9]];
    CONST robtarget p3801:= [[1500.8038916021112, 55.58661703595381, 993.500033578516], [0, 0, 1, 0], [0, 0, 0, 0], [9E9, 9E9, 9E9, 9E9, 9E9, 9E9]];
    CONST robtarget p3802:= [[1501.0716136418002, 55.58179702378129, 993.500033578516], [0, 0, 1, 0], [0, 0, 0, 0], [9E9, 9E9, 9E9, 9E9, 9E9, 9E9]];
    CONST robtarget p3803:= [[1501.4777166673434, 55.58716507590418, 993.500033578516], [0, 0, 1, 0], [0, 0, 0, 0], [9E9, 9E9, 9E9, 9E9, 9E9, 9E9]];
    CONST robtarget p3804:= [[1501.74986056141, 55.57291410341341, 993.500033578516], [0, 0, 1, 0], [0, 0, 0, 0], [9E9, 9E9, 9E9, 9E9, 9E9, 9E9]];
    CONST robtarget p3805:= [[1502.508235227333, 55.54892422779126, 993.500033578516], [0, 0, 1, 0], [0, 0, 0, 0], [9E9, 9E9, 9E9, 9E9, 9E9, 9E9]];
    CONST robtarget p3806:= [[1502.7718201424705, 55.53306216926774, 993.500033578516], [0, 0, 1, 0], [0, 0, 0, 0], [9E9, 9E9, 9E9, 9E9, 9E9, 9E9]];
    CONST robtarget p3807:= [[1503.1591981760482, 55.49833530965907, 993.500033578516], [0, 0, 1, 0], [0, 0, 0, 0], [9E9, 9E9, 9E9, 9E9, 9E9, 9E9]];
    CONST robtarget p3808:= [[1503.529519604504, 55.468994956774765, 993.500033578516], [0, 0, 1, 0], [0, 0, 0, 0], [9E9, 9E9, 9E9, 9E9, 9E9, 9E9]];
    CONST robtarget p3809:= [[1503.9027279836116, 55.44585318494282, 993.500033578516], [0, 0, 1, 0], [0, 0, 0, 0], [9E9, 9E9, 9E9, 9E9, 9E9, 9E9]];
    CONST robtarget p3810:= [[1504.1305203451661, 55.420657230435964, 993.500033578516], [0, 0, 1, 0], [0, 0, 0, 0], [9E9, 9E9, 9E9, 9E9, 9E9, 9E9]];
    CONST robtarget p3811:= [[1504.45370942973, 55.399988632971, 993.500033578516], [0, 0, 1, 0], [0, 0, 0, 0], [9E9, 9E9, 9E9, 9E9, 9E9, 9E9]];
    CONST robtarget p3812:= [[1504.8692542553433, 55.37165906033243, 993.500033578516], [0, 0, 1, 0], [0, 0, 0, 0], [9E9, 9E9, 9E9, 9E9, 9E9, 9E9]];
    CONST robtarget p3813:= [[1505.213123493795, 55.34129281481901, 993.500033578516], [0, 0, 1, 0], [0, 0, 0, 0], [9E9, 9E9, 9E9, 9E9, 9E9, 9E9]];
    CONST robtarget p3814:= [[1505.5487829320978, 55.311295760649315, 993.500033578516], [0, 0, 1, 0], [0, 0, 0, 0], [9E9, 9E9, 9E9, 9E9, 9E9, 9E9]];
    CONST robtarget p3815:= [[1505.872186890476, 55.29324398698951, 993.500033578516], [0, 0, 1, 0], [0, 0, 0, 0], [9E9, 9E9, 9E9, 9E9, 9E9, 9E9]];
    CONST robtarget p3816:= [[1506.1069429683735, 55.28041096681888, 993.500033578516], [0, 0, 1, 0], [0, 0, 0, 0], [9E9, 9E9, 9E9, 9E9, 9E9, 9E9]];
    CONST robtarget p3817:= [[1506.2175886136542, 55.26351352331109, 993.500033578516], [0, 0, 1, 0], [0, 0, 0, 0], [9E9, 9E9, 9E9, 9E9, 9E9, 9E9]];
    CONST robtarget p3818:= [[1506.4083010887966, 55.23181883321082, 993.500033578516], [0, 0, 1, 0], [0, 0, 0, 0], [9E9, 9E9, 9E9, 9E9, 9E9, 9E9]];
    CONST robtarget p3819:= [[1507.032788328069, 55.15019966174758, 993.500033578516], [0, 0, 1, 0], [0, 0, 0, 0], [9E9, 9E9, 9E9, 9E9, 9E9, 9E9]];
    CONST robtarget p3820:= [[1507.3639393909004, 55.09170701741259, 993.500033578516], [0, 0, 1, 0], [0, 0, 0, 0], [9E9, 9E9, 9E9, 9E9, 9E9, 9E9]];
    CONST robtarget p3821:= [[1507.7735057730338, 55.03572699825082, 993.500033578516], [0, 0, 1, 0], [0, 0, 0, 0], [9E9, 9E9, 9E9, 9E9, 9E9, 9E9]];
    CONST robtarget p3822:= [[1508.5061765994722, 54.92556586810123, 993.500033578516], [0, 0, 1, 0], [0, 0, 0, 0], [9E9, 9E9, 9E9, 9E9, 9E9, 9E9]];
    CONST robtarget p3823:= [[1508.5633269766688, 54.92039239510473, 993.500033578516], [0, 0, 1, 0], [0, 0, 0, 0], [9E9, 9E9, 9E9, 9E9, 9E9, 9E9]];
    CONST robtarget p3824:= [[1508.6871471675622, 54.90140191916876, 993.500033578516], [0, 0, 1, 0], [0, 0, 0, 0], [9E9, 9E9, 9E9, 9E9, 9E9, 9E9]];
    CONST robtarget p3825:= [[1509.111528640207, 54.839146628118954, 993.500033578516], [0, 0, 1, 0], [0, 0, 0, 0], [9E9, 9E9, 9E9, 9E9, 9E9, 9E9]];
    CONST robtarget p3826:= [[1509.5658185340976, 54.77790933467254, 993.500033578516], [0, 0, 1, 0], [0, 0, 0, 0], [9E9, 9E9, 9E9, 9E9, 9E9, 9E9]];
    CONST robtarget p3827:= [[1509.719834375291, 54.74988978690848, 993.500033578516], [0, 0, 1, 0], [0, 0, 0, 0], [9E9, 9E9, 9E9, 9E9, 9E9, 9E9]];
    CONST robtarget p3828:= [[1510.2327532778063, 54.66681359100322, 993.500033578516], [0, 0, 1, 0], [0, 0, 0, 0], [9E9, 9E9, 9E9, 9E9, 9E9, 9E9]];
    CONST robtarget p3829:= [[1510.708285403098, 54.54912181192752, 993.500033578516], [0, 0, 1, 0], [0, 0, 0, 0], [9E9, 9E9, 9E9, 9E9, 9E9, 9E9]];
    CONST robtarget p3830:= [[1510.9871551635622, 54.492475199660745, 993.500033578516], [0, 0, 1, 0], [0, 0, 0, 0], [9E9, 9E9, 9E9, 9E9, 9E9, 9E9]];
    CONST robtarget p3831:= [[1511.2139798826, 54.45038870208272, 993.500033578516], [0, 0, 1, 0], [0, 0, 0, 0], [9E9, 9E9, 9E9, 9E9, 9E9, 9E9]];
    CONST robtarget p3832:= [[1511.7068679335039, 54.327043949393484, 993.500033578516], [0, 0, 1, 0], [0, 0, 0, 0], [9E9, 9E9, 9E9, 9E9, 9E9, 9E9]];
    CONST robtarget p3833:= [[1511.9542442231402, 54.28121262053381, 993.500033578516], [0, 0, 1, 0], [0, 0, 0, 0], [9E9, 9E9, 9E9, 9E9, 9E9, 9E9]];
    CONST robtarget p3834:= [[1512.1123556892765, 54.24884802163942, 993.500033578516], [0, 0, 1, 0], [0, 0, 0, 0], [9E9, 9E9, 9E9, 9E9, 9E9, 9E9]];
    CONST robtarget p3835:= [[1512.4640320696003, 54.16405290260806, 993.500033578516], [0, 0, 1, 0], [0, 0, 0, 0], [9E9, 9E9, 9E9, 9E9, 9E9, 9E9]];
    CONST robtarget p3836:= [[1512.9885205244661, 54.04383941848825, 993.500033578516], [0, 0, 1, 0], [0, 0, 0, 0], [9E9, 9E9, 9E9, 9E9, 9E9, 9E9]];
    CONST robtarget p3837:= [[1513.4699361972723, 53.92842011643258, 993.500033578516], [0, 0, 1, 0], [0, 0, 0, 0], [9E9, 9E9, 9E9, 9E9, 9E9, 9E9]];
    CONST robtarget p3838:= [[1514.209809429855, 53.76446442876235, 993.500033578516], [0, 0, 1, 0], [0, 0, 0, 0], [9E9, 9E9, 9E9, 9E9, 9E9, 9E9]];
    CONST robtarget p3839:= [[1514.4510141491096, 53.687943367027984, 993.500033578516], [0, 0, 1, 0], [0, 0, 0, 0], [9E9, 9E9, 9E9, 9E9, 9E9, 9E9]];
    CONST robtarget p3840:= [[1514.6502997450727, 53.634448642732806, 993.500033578516], [0, 0, 1, 0], [0, 0, 0, 0], [9E9, 9E9, 9E9, 9E9, 9E9, 9E9]];
    CONST robtarget p3841:= [[1514.919996655769, 53.545010846360725, 993.500033578516], [0, 0, 1, 0], [0, 0, 0, 0], [9E9, 9E9, 9E9, 9E9, 9E9, 9E9]];
    CONST robtarget p3842:= [[1515.2779485200285, 53.436491611333636, 993.500033578516], [0, 0, 1, 0], [0, 0, 0, 0], [9E9, 9E9, 9E9, 9E9, 9E9, 9E9]];
    CONST robtarget p3843:= [[1515.4945755008719, 53.37396207703124, 993.500033578516], [0, 0, 1, 0], [0, 0, 0, 0], [9E9, 9E9, 9E9, 9E9, 9E9, 9E9]];
    CONST robtarget p3844:= [[1515.7235409640637, 53.31074968429867, 993.500033578516], [0, 0, 1, 0], [0, 0, 0, 0], [9E9, 9E9, 9E9, 9E9, 9E9, 9E9]];
    CONST robtarget p3845:= [[1515.9951132737951, 53.22485876665587, 993.500033578516], [0, 0, 1, 0], [0, 0, 0, 0], [9E9, 9E9, 9E9, 9E9, 9E9, 9E9]];
    CONST robtarget p3846:= [[1516.5286130051163, 53.06742443896117, 993.500033578516], [0, 0, 1, 0], [0, 0, 0, 0], [9E9, 9E9, 9E9, 9E9, 9E9, 9E9]];
    CONST robtarget p3847:= [[1517.1147361152496, 52.883824263349126, 993.500033578516], [0, 0, 1, 0], [0, 0, 0, 0], [9E9, 9E9, 9E9, 9E9, 9E9, 9E9]];
    CONST robtarget p3848:= [[1517.5157962468943, 52.77194953767355, 993.500033578516], [0, 0, 1, 0], [0, 0, 0, 0], [9E9, 9E9, 9E9, 9E9, 9E9, 9E9]];
    CONST robtarget p3849:= [[1517.7729613911822, 52.69725496137872, 993.500033578516], [0, 0, 1, 0], [0, 0, 0, 0], [9E9, 9E9, 9E9, 9E9, 9E9, 9E9]];
    CONST robtarget p3850:= [[1518.3122321678754, 52.49840204464448, 993.500033578516], [0, 0, 1, 0], [0, 0, 0, 0], [9E9, 9E9, 9E9, 9E9, 9E9, 9E9]];
    CONST robtarget p3851:= [[1518.8327709357088, 52.291441343989746, 993.500033578516], [0, 0, 1, 0], [0, 0, 0, 0], [9E9, 9E9, 9E9, 9E9, 9E9, 9E9]];
    CONST robtarget p3852:= [[1519.2327430619562, 52.156244292877204, 993.500033578516], [0, 0, 1, 0], [0, 0, 0, 0], [9E9, 9E9, 9E9, 9E9, 9E9, 9E9]];
    CONST robtarget p3853:= [[1519.4652154180876, 52.058936917535576, 993.500033578516], [0, 0, 1, 0], [0, 0, 0, 0], [9E9, 9E9, 9E9, 9E9, 9E9, 9E9]];
    CONST robtarget p3854:= [[1519.9666097868185, 51.873894197107376, 993.500033578516], [0, 0, 1, 0], [0, 0, 0, 0], [9E9, 9E9, 9E9, 9E9, 9E9, 9E9]];
    CONST robtarget p3855:= [[1520.1357073901772, 51.80243252868593, 993.500033578516], [0, 0, 1, 0], [0, 0, 0, 0], [9E9, 9E9, 9E9, 9E9, 9E9, 9E9]];
    CONST robtarget p3856:= [[1520.4967786102009, 51.66563949693334, 993.500033578516], [0, 0, 1, 0], [0, 0, 0, 0], [9E9, 9E9, 9E9, 9E9, 9E9, 9E9]];
    CONST robtarget p3857:= [[1520.7569566228976, 51.571982723733626, 993.500033578516], [0, 0, 1, 0], [0, 0, 0, 0], [9E9, 9E9, 9E9, 9E9, 9E9, 9E9]];
    CONST robtarget p3858:= [[1521.020149949859, 51.46809113856294, 993.500033578516], [0, 0, 1, 0], [0, 0, 0, 0], [9E9, 9E9, 9E9, 9E9, 9E9, 9E9]];
    CONST robtarget p3859:= [[1521.1878954550139, 51.403043598968196, 993.500033578516], [0, 0, 1, 0], [0, 0, 0, 0], [9E9, 9E9, 9E9, 9E9, 9E9, 9E9]];
    CONST robtarget p3860:= [[1521.365337984672, 51.3394427502071, 993.500033578516], [0, 0, 1, 0], [0, 0, 0, 0], [9E9, 9E9, 9E9, 9E9, 9E9, 9E9]];
    CONST robtarget p3861:= [[1521.6925120940898, 51.20431425468752, 993.500033578516], [0, 0, 1, 0], [0, 0, 0, 0], [9E9, 9E9, 9E9, 9E9, 9E9, 9E9]];
    CONST robtarget p3862:= [[1521.7904058627012, 51.1589171680678, 993.500033578516], [0, 0, 1, 0], [0, 0, 0, 0], [9E9, 9E9, 9E9, 9E9, 9E9, 9E9]];
    CONST robtarget p3863:= [[1522.059408955089, 51.027137934123985, 993.500033578516], [0, 0, 1, 0], [0, 0, 0, 0], [9E9, 9E9, 9E9, 9E9, 9E9, 9E9]];
    CONST robtarget p3864:= [[1522.2229877357165, 50.95182741555061, 993.500033578516], [0, 0, 1, 0], [0, 0, 0, 0], [9E9, 9E9, 9E9, 9E9, 9E9, 9E9]];
    CONST robtarget p3865:= [[1522.4991510178022, 50.82827136348807, 993.500033578516], [0, 0, 1, 0], [0, 0, 0, 0], [9E9, 9E9, 9E9, 9E9, 9E9, 9E9]];
    CONST robtarget p3866:= [[1522.7721307284999, 50.712636979107714, 993.500033578516], [0, 0, 1, 0], [0, 0, 0, 0], [9E9, 9E9, 9E9, 9E9, 9E9, 9E9]];
    CONST robtarget p3867:= [[1522.9452226855071, 50.63308094179159, 993.500033578516], [0, 0, 1, 0], [0, 0, 0, 0], [9E9, 9E9, 9E9, 9E9, 9E9, 9E9]];
    CONST robtarget p3868:= [[1523.3662050647742, 50.426821451896515, 993.500033578516], [0, 0, 1, 0], [0, 0, 0, 0], [9E9, 9E9, 9E9, 9E9, 9E9, 9E9]];
    CONST robtarget p3869:= [[1523.5904115480603, 50.32011418543033, 993.500033578516], [0, 0, 1, 0], [0, 0, 0, 0], [9E9, 9E9, 9E9, 9E9, 9E9, 9E9]];
    CONST robtarget p3870:= [[1524.2199501573416, 50.0219833799905, 993.500033578516], [0, 0, 1, 0], [0, 0, 0, 0], [9E9, 9E9, 9E9, 9E9, 9E9, 9E9]];
    CONST robtarget p3871:= [[1524.6265463564314, 49.823761052554886, 993.500033578516], [0, 0, 1, 0], [0, 0, 0, 0], [9E9, 9E9, 9E9, 9E9, 9E9, 9E9]];
    CONST robtarget p3872:= [[1524.8633929743323, 49.72834275828113, 993.500033578516], [0, 0, 1, 0], [0, 0, 0, 0], [9E9, 9E9, 9E9, 9E9, 9E9, 9E9]];
    CONST robtarget p3873:= [[1524.9225158081774, 49.699785499267776, 993.500033578516], [0, 0, 1, 0], [0, 0, 0, 0], [9E9, 9E9, 9E9, 9E9, 9E9, 9E9]];
    CONST robtarget p3874:= [[1525.2971317852357, 49.5162665236673, 993.500033578516], [0, 0, 1, 0], [0, 0, 0, 0], [9E9, 9E9, 9E9, 9E9, 9E9, 9E9]];
    CONST robtarget p3875:= [[1525.6868004111063, 49.31630559969699, 993.500033578516], [0, 0, 1, 0], [0, 0, 0, 0], [9E9, 9E9, 9E9, 9E9, 9E9, 9E9]];
    CONST robtarget p3876:= [[1526.0815794428704, 49.10279898035205, 993.500033578516], [0, 0, 1, 0], [0, 0, 0, 0], [9E9, 9E9, 9E9, 9E9, 9E9, 9E9]];
    CONST robtarget p3877:= [[1526.3760813943888, 48.93726623406556, 993.500033578516], [0, 0, 1, 0], [0, 0, 0, 0], [9E9, 9E9, 9E9, 9E9, 9E9, 9E9]];
    CONST robtarget p3878:= [[1526.7870042397735, 48.7026507291059, 993.500033578516], [0, 0, 1, 0], [0, 0, 0, 0], [9E9, 9E9, 9E9, 9E9, 9E9, 9E9]];
    CONST robtarget p3879:= [[1527.1230931951618, 48.508693069278095, 993.500033578516], [0, 0, 1, 0], [0, 0, 0, 0], [9E9, 9E9, 9E9, 9E9, 9E9, 9E9]];
    CONST robtarget p3880:= [[1527.58317110616, 48.24630642461811, 993.500033578516], [0, 0, 1, 0], [0, 0, 0, 0], [9E9, 9E9, 9E9, 9E9, 9E9, 9E9]];
    CONST robtarget p3881:= [[1527.7113238345817, 48.18337831288005, 993.500033578516], [0, 0, 1, 0], [0, 0, 0, 0], [9E9, 9E9, 9E9, 9E9, 9E9, 9E9]];
    CONST robtarget p3882:= [[1527.8198690160962, 48.11957965009027, 993.500033578516], [0, 0, 1, 0], [0, 0, 0, 0], [9E9, 9E9, 9E9, 9E9, 9E9, 9E9]];
    CONST robtarget p3883:= [[1528.1569667893164, 47.92386918244411, 993.500033578516], [0, 0, 1, 0], [0, 0, 0, 0], [9E9, 9E9, 9E9, 9E9, 9E9, 9E9]];
    CONST robtarget p3884:= [[1528.313032532701, 47.84024766233027, 993.500033578516], [0, 0, 1, 0], [0, 0, 0, 0], [9E9, 9E9, 9E9, 9E9, 9E9, 9E9]];
    CONST robtarget p3885:= [[1528.5597902838576, 47.70678584687879, 993.500033578516], [0, 0, 1, 0], [0, 0, 0, 0], [9E9, 9E9, 9E9, 9E9, 9E9, 9E9]];
    CONST robtarget p3886:= [[1528.9757197829558, 47.470989939424214, 993.500033578516], [0, 0, 1, 0], [0, 0, 0, 0], [9E9, 9E9, 9E9, 9E9, 9E9, 9E9]];
    CONST robtarget p3887:= [[1529.0790509044512, 47.40243258482579, 993.500033578516], [0, 0, 1, 0], [0, 0, 0, 0], [9E9, 9E9, 9E9, 9E9, 9E9, 9E9]];
    CONST robtarget p3888:= [[1529.2674697416405, 47.27242684039334, 993.500033578516], [0, 0, 1, 0], [0, 0, 0, 0], [9E9, 9E9, 9E9, 9E9, 9E9, 9E9]];
    CONST robtarget p3889:= [[1529.8493466113212, 46.889890372526764, 993.500033578516], [0, 0, 1, 0], [0, 0, 0, 0], [9E9, 9E9, 9E9, 9E9, 9E9, 9E9]];
    CONST robtarget p3890:= [[1530.0491625353816, 46.75095021961015, 993.500033578516], [0, 0, 1, 0], [0, 0, 0, 0], [9E9, 9E9, 9E9, 9E9, 9E9, 9E9]];
    CONST robtarget p3891:= [[1530.613330919521, 46.393355648391434, 993.500033578516], [0, 0, 1, 0], [0, 0, 0, 0], [9E9, 9E9, 9E9, 9E9, 9E9, 9E9]];
    CONST robtarget p3892:= [[1530.795630304955, 46.268604669387685, 993.500033578516], [0, 0, 1, 0], [0, 0, 0, 0], [9E9, 9E9, 9E9, 9E9, 9E9, 9E9]];
    CONST robtarget p3893:= [[1531.344372084039, 45.897625377020645, 993.500033578516], [0, 0, 1, 0], [0, 0, 0, 0], [9E9, 9E9, 9E9, 9E9, 9E9, 9E9]];
    CONST robtarget p3894:= [[1531.7851458773612, 45.61801771916723, 993.500033578516], [0, 0, 1, 0], [0, 0, 0, 0], [9E9, 9E9, 9E9, 9E9, 9E9, 9E9]];
    CONST robtarget p3895:= [[1532.1416508338064, 45.37846692249079, 993.500033578516], [0, 0, 1, 0], [0, 0, 0, 0], [9E9, 9E9, 9E9, 9E9, 9E9, 9E9]];
    CONST robtarget p3896:= [[1532.3071133848148, 45.26059154304093, 993.500033578516], [0, 0, 1, 0], [0, 0, 0, 0], [9E9, 9E9, 9E9, 9E9, 9E9, 9E9]];
    CONST robtarget p3897:= [[1532.5205539558342, 45.10802654210809, 993.500033578516], [0, 0, 1, 0], [0, 0, 0, 0], [9E9, 9E9, 9E9, 9E9, 9E9, 9E9]];
    CONST robtarget p3898:= [[1532.8427088142992, 44.85476638754251, 993.500033578516], [0, 0, 1, 0], [0, 0, 0, 0], [9E9, 9E9, 9E9, 9E9, 9E9, 9E9]];
    CONST robtarget p3899:= [[1533.036006499551, 44.71714222835308, 993.500033578516], [0, 0, 1, 0], [0, 0, 0, 0], [9E9, 9E9, 9E9, 9E9, 9E9, 9E9]];
    CONST robtarget p3900:= [[1533.2794732126126, 44.52447366543173, 993.500033578516], [0, 0, 1, 0], [0, 0, 0, 0], [9E9, 9E9, 9E9, 9E9, 9E9, 9E9]];
    CONST robtarget p3901:= [[1533.372108252455, 44.4516796110636, 993.500033578516], [0, 0, 1, 0], [0, 0, 0, 0], [9E9, 9E9, 9E9, 9E9, 9E9, 9E9]];
    CONST robtarget p3902:= [[1533.956690252653, 43.99466469693871, 993.500033578516], [0, 0, 1, 0], [0, 0, 0, 0], [9E9, 9E9, 9E9, 9E9, 9E9, 9E9]];
    CONST robtarget p3903:= [[1534.2923623823035, 43.744139333967325, 993.500033578516], [0, 0, 1, 0], [0, 0, 0, 0], [9E9, 9E9, 9E9, 9E9, 9E9, 9E9]];
    CONST robtarget p3904:= [[1534.4508477024613, 43.620365943949395, 993.500033578516], [0, 0, 1, 0], [0, 0, 0, 0], [9E9, 9E9, 9E9, 9E9, 9E9, 9E9]];
    CONST robtarget p3905:= [[1534.8835771222748, 43.28252363985814, 993.500033578516], [0, 0, 1, 0], [0, 0, 0, 0], [9E9, 9E9, 9E9, 9E9, 9E9, 9E9]];
    CONST robtarget p3906:= [[1535.0188902871541, 43.16951504045551, 993.500033578516], [0, 0, 1, 0], [0, 0, 0, 0], [9E9, 9E9, 9E9, 9E9, 9E9, 9E9]];
    CONST robtarget p3907:= [[1535.3297049402547, 42.92796242797951, 993.500033578516], [0, 0, 1, 0], [0, 0, 0, 0], [9E9, 9E9, 9E9, 9E9, 9E9, 9E9]];
    CONST robtarget p3908:= [[1535.6392921168788, 42.69850257901318, 993.500033578516], [0, 0, 1, 0], [0, 0, 0, 0], [9E9, 9E9, 9E9, 9E9, 9E9, 9E9]];
    CONST robtarget p3909:= [[1536.0629564778342, 42.318671823519054, 993.500033578516], [0, 0, 1, 0], [0, 0, 0, 0], [9E9, 9E9, 9E9, 9E9, 9E9, 9E9]];
    CONST robtarget p3910:= [[1536.2154924297377, 42.18294208118489, 993.500033578516], [0, 0, 1, 0], [0, 0, 0, 0], [9E9, 9E9, 9E9, 9E9, 9E9, 9E9]];
    CONST robtarget p3911:= [[1536.275214853649, 42.12888861013877, 993.500033578516], [0, 0, 1, 0], [0, 0, 0, 0], [9E9, 9E9, 9E9, 9E9, 9E9, 9E9]];
    CONST robtarget p3912:= [[1536.3536973007845, 42.05412139537343, 993.500033578516], [0, 0, 1, 0], [0, 0, 0, 0], [9E9, 9E9, 9E9, 9E9, 9E9, 9E9]];
    CONST robtarget p3913:= [[1536.5114415599312, 41.91258406937128, 993.500033578516], [0, 0, 1, 0], [0, 0, 0, 0], [9E9, 9E9, 9E9, 9E9, 9E9, 9E9]];
    CONST robtarget p3914:= [[1536.9066644569052, 41.537868758763665, 993.500033578516], [0, 0, 1, 0], [0, 0, 0, 0], [9E9, 9E9, 9E9, 9E9, 9E9, 9E9]];
    CONST robtarget p3915:= [[1537.1702523366748, 41.307557916758654, 993.500033578516], [0, 0, 1, 0], [0, 0, 0, 0], [9E9, 9E9, 9E9, 9E9, 9E9, 9E9]];
    CONST robtarget p3916:= [[1537.2790121547498, 41.21242337742689, 993.500033578516], [0, 0, 1, 0], [0, 0, 0, 0], [9E9, 9E9, 9E9, 9E9, 9E9, 9E9]];
    CONST robtarget p3917:= [[1537.5430743042257, 40.98646395752229, 993.500033578516], [0, 0, 1, 0], [0, 0, 0, 0], [9E9, 9E9, 9E9, 9E9, 9E9, 9E9]];
    CONST robtarget p3918:= [[1537.7054780186418, 40.83509144678578, 993.500033578516], [0, 0, 1, 0], [0, 0, 0, 0], [9E9, 9E9, 9E9, 9E9, 9E9, 9E9]];
    CONST robtarget p3919:= [[1537.938039252857, 40.638829683634924, 993.500033578516], [0, 0, 1, 0], [0, 0, 0, 0], [9E9, 9E9, 9E9, 9E9, 9E9, 9E9]];
    CONST robtarget p3920:= [[1538.4965751958885, 40.13545271275093, 993.500033578516], [0, 0, 1, 0], [0, 0, 0, 0], [9E9, 9E9, 9E9, 9E9, 9E9, 9E9]];
    CONST robtarget p3921:= [[1538.8767089701246, 39.74447345553044, 993.500033578516], [0, 0, 1, 0], [0, 0, 0, 0], [9E9, 9E9, 9E9, 9E9, 9E9, 9E9]];
    CONST robtarget p3922:= [[1539.0969797847454, 39.52951611463887, 993.500033578516], [0, 0, 1, 0], [0, 0, 0, 0], [9E9, 9E9, 9E9, 9E9, 9E9, 9E9]];
    CONST robtarget p3923:= [[1539.1991512084876, 39.41464714768044, 993.500033578516], [0, 0, 1, 0], [0, 0, 0, 0], [9E9, 9E9, 9E9, 9E9, 9E9, 9E9]];
    CONST robtarget p3924:= [[1539.4365277593558, 39.151146986042534, 993.500033578516], [0, 0, 1, 0], [0, 0, 0, 0], [9E9, 9E9, 9E9, 9E9, 9E9, 9E9]];
    CONST robtarget p3925:= [[1539.7742949108756, 38.79295618787974, 993.500033578516], [0, 0, 1, 0], [0, 0, 0, 0], [9E9, 9E9, 9E9, 9E9, 9E9, 9E9]];
    CONST robtarget p3926:= [[1539.9759767634803, 38.593596628757055, 993.500033578516], [0, 0, 1, 0], [0, 0, 0, 0], [9E9, 9E9, 9E9, 9E9, 9E9, 9E9]];
    CONST robtarget p3927:= [[1540.2182239790054, 38.365419043027615, 993.500033578516], [0, 0, 1, 0], [0, 0, 0, 0], [9E9, 9E9, 9E9, 9E9, 9E9, 9E9]];
    CONST robtarget p3928:= [[1540.5269553637595, 38.04203469863677, 993.500033578516], [0, 0, 1, 0], [0, 0, 0, 0], [9E9, 9E9, 9E9, 9E9, 9E9, 9E9]];
    CONST robtarget p3929:= [[1540.7922750766197, 37.77284763027346, 993.500033578516], [0, 0, 1, 0], [0, 0, 0, 0], [9E9, 9E9, 9E9, 9E9, 9E9, 9E9]];
    CONST robtarget p3930:= [[1541.028127903321, 37.519033820117016, 993.500033578516], [0, 0, 1, 0], [0, 0, 0, 0], [9E9, 9E9, 9E9, 9E9, 9E9, 9E9]];
    CONST robtarget p3931:= [[1541.2372982553477, 37.30729757697519, 993.500033578516], [0, 0, 1, 0], [0, 0, 0, 0], [9E9, 9E9, 9E9, 9E9, 9E9, 9E9]];
    CONST robtarget p3932:= [[1541.5308646062183, 36.963007780385794, 993.500033578516], [0, 0, 1, 0], [0, 0, 0, 0], [9E9, 9E9, 9E9, 9E9, 9E9, 9E9]];
    CONST robtarget p3933:= [[1541.8108772005746, 36.649499215957576, 993.500033578516], [0, 0, 1, 0], [0, 0, 0, 0], [9E9, 9E9, 9E9, 9E9, 9E9, 9E9]];
    CONST robtarget p3934:= [[1542.1927195344256, 36.19139843511296, 993.500033578516], [0, 0, 1, 0], [0, 0, 0, 0], [9E9, 9E9, 9E9, 9E9, 9E9, 9E9]];
    CONST robtarget p3935:= [[1542.4420005783538, 35.892081418588035, 993.500033578516], [0, 0, 1, 0], [0, 0, 0, 0], [9E9, 9E9, 9E9, 9E9, 9E9, 9E9]];
    CONST robtarget p3936:= [[1542.7611487073411, 35.49913467927132, 993.500033578516], [0, 0, 1, 0], [0, 0, 0, 0], [9E9, 9E9, 9E9, 9E9, 9E9, 9E9]];
    CONST robtarget p3937:= [[1542.9359534249188, 35.29474336046775, 993.500033578516], [0, 0, 1, 0], [0, 0, 0, 0], [9E9, 9E9, 9E9, 9E9, 9E9, 9E9]];
    CONST robtarget p3938:= [[1543.1076606594088, 35.08643507015543, 993.500033578516], [0, 0, 1, 0], [0, 0, 0, 0], [9E9, 9E9, 9E9, 9E9, 9E9, 9E9]];
    CONST robtarget p3939:= [[1543.2371478590371, 34.92046676462293, 993.500033578516], [0, 0, 1, 0], [0, 0, 0, 0], [9E9, 9E9, 9E9, 9E9, 9E9, 9E9]];
    CONST robtarget p3940:= [[1543.5154969815137, 34.58113324901245, 993.500033578516], [0, 0, 1, 0], [0, 0, 0, 0], [9E9, 9E9, 9E9, 9E9, 9E9, 9E9]];
    CONST robtarget p3941:= [[1543.7222098969098, 34.34229844079741, 993.500033578516], [0, 0, 1, 0], [0, 0, 0, 0], [9E9, 9E9, 9E9, 9E9, 9E9, 9E9]];
    CONST robtarget p3942:= [[1543.946405024249, 34.05550196223993, 993.500033578516], [0, 0, 1, 0], [0, 0, 0, 0], [9E9, 9E9, 9E9, 9E9, 9E9, 9E9]];
    CONST robtarget p3943:= [[1544.3591772107966, 33.5160521331772, 993.500033578516], [0, 0, 1, 0], [0, 0, 0, 0], [9E9, 9E9, 9E9, 9E9, 9E9, 9E9]];
    CONST robtarget p3944:= [[1544.6918058715369, 33.03983782569199, 993.500033578516], [0, 0, 1, 0], [0, 0, 0, 0], [9E9, 9E9, 9E9, 9E9, 9E9, 9E9]];
    CONST robtarget p3945:= [[1544.9187768956888, 32.73271957089845, 993.500033578516], [0, 0, 1, 0], [0, 0, 0, 0], [9E9, 9E9, 9E9, 9E9, 9E9, 9E9]];
    CONST robtarget p3946:= [[1545.0282166349157, 32.58822388497079, 993.500033578516], [0, 0, 1, 0], [0, 0, 0, 0], [9E9, 9E9, 9E9, 9E9, 9E9, 9E9]];
    CONST robtarget p3947:= [[1545.1287786360754, 32.44827758234318, 993.500033578516], [0, 0, 1, 0], [0, 0, 0, 0], [9E9, 9E9, 9E9, 9E9, 9E9, 9E9]];
    CONST robtarget p3948:= [[1545.4545830833977, 31.986822350448634, 993.500033578516], [0, 0, 1, 0], [0, 0, 0, 0], [9E9, 9E9, 9E9, 9E9, 9E9, 9E9]];
    CONST robtarget p3949:= [[1545.6703457364565, 31.687875094378597, 993.500033578516], [0, 0, 1, 0], [0, 0, 0, 0], [9E9, 9E9, 9E9, 9E9, 9E9, 9E9]];
    CONST robtarget p3950:= [[1545.968873789536, 31.246618912589398, 993.500033578516], [0, 0, 1, 0], [0, 0, 0, 0], [9E9, 9E9, 9E9, 9E9, 9E9, 9E9]];
    CONST robtarget p3951:= [[1546.1838561632724, 30.958378163329954, 993.500033578516], [0, 0, 1, 0], [0, 0, 0, 0], [9E9, 9E9, 9E9, 9E9, 9E9, 9E9]];
    CONST robtarget p3952:= [[1546.2743750338382, 30.843870698332736, 993.500033578516], [0, 0, 1, 0], [0, 0, 0, 0], [9E9, 9E9, 9E9, 9E9, 9E9, 9E9]];
    CONST robtarget p3953:= [[1546.4102251639426, 30.639047610340896, 993.500033578516], [0, 0, 1, 0], [0, 0, 0, 0], [9E9, 9E9, 9E9, 9E9, 9E9, 9E9]];
    CONST robtarget p3954:= [[1546.631452559879, 30.259468304842116, 993.500033578516], [0, 0, 1, 0], [0, 0, 0, 0], [9E9, 9E9, 9E9, 9E9, 9E9, 9E9]];
    CONST robtarget p3955:= [[1546.8103666461084, 29.980076615591017, 993.500033578516], [0, 0, 1, 0], [0, 0, 0, 0], [9E9, 9E9, 9E9, 9E9, 9E9, 9E9]];
    CONST robtarget p3956:= [[1547.056173845242, 29.584456861448672, 993.500033578516], [0, 0, 1, 0], [0, 0, 0, 0], [9E9, 9E9, 9E9, 9E9, 9E9, 9E9]];
    CONST robtarget p3957:= [[1547.1132431492347, 29.49214410705595, 993.500033578516], [0, 0, 1, 0], [0, 0, 0, 0], [9E9, 9E9, 9E9, 9E9, 9E9, 9E9]];
    CONST robtarget p3958:= [[1547.2242215028514, 29.29043977930145, 993.500033578516], [0, 0, 1, 0], [0, 0, 0, 0], [9E9, 9E9, 9E9, 9E9, 9E9, 9E9]];
    CONST robtarget p3959:= [[1547.5542971895707, 28.775112930323772, 993.500033578516], [0, 0, 1, 0], [0, 0, 0, 0], [9E9, 9E9, 9E9, 9E9, 9E9, 9E9]];
    CONST robtarget p3960:= [[1547.8142917521911, 28.335989704485883, 993.500033578516], [0, 0, 1, 0], [0, 0, 0, 0], [9E9, 9E9, 9E9, 9E9, 9E9, 9E9]];
    CONST robtarget p3961:= [[1547.9376784976303, 28.14314913169777, 993.500033578516], [0, 0, 1, 0], [0, 0, 0, 0], [9E9, 9E9, 9E9, 9E9, 9E9, 9E9]];
    CONST robtarget p3962:= [[1548.2983833854353, 27.543577638096295, 993.500033578516], [0, 0, 1, 0], [0, 0, 0, 0], [9E9, 9E9, 9E9, 9E9, 9E9, 9E9]];
    CONST robtarget p3963:= [[1548.3628428745214, 27.44770545310911, 993.500033578516], [0, 0, 1, 0], [0, 0, 0, 0], [9E9, 9E9, 9E9, 9E9, 9E9, 9E9]];
    CONST robtarget p3964:= [[1548.43394074674, 27.323574898397794, 993.500033578516], [0, 0, 1, 0], [0, 0, 0, 0], [9E9, 9E9, 9E9, 9E9, 9E9, 9E9]];
    CONST robtarget p3965:= [[1548.628655854489, 26.965269518030638, 993.500033578516], [0, 0, 1, 0], [0, 0, 0, 0], [9E9, 9E9, 9E9, 9E9, 9E9, 9E9]];
    CONST robtarget p3966:= [[1548.6483106899937, 26.922131624905774, 993.500033578516], [0, 0, 1, 0], [0, 0, 0, 0], [9E9, 9E9, 9E9, 9E9, 9E9, 9E9]];
    CONST robtarget p3967:= [[1548.783397038658, 26.64113542049482, 993.500033578516], [0, 0, 1, 0], [0, 0, 0, 0], [9E9, 9E9, 9E9, 9E9, 9E9, 9E9]];
    CONST robtarget p3968:= [[1548.9188277190328, 26.35081169788687, 993.500033578516], [0, 0, 1, 0], [0, 0, 0, 0], [9E9, 9E9, 9E9, 9E9, 9E9, 9E9]];
    CONST robtarget p3969:= [[1549.2395290852285, 25.783503588668964, 993.500033578516], [0, 0, 1, 0], [0, 0, 0, 0], [9E9, 9E9, 9E9, 9E9, 9E9, 9E9]];
    CONST robtarget p3970:= [[1549.5622838212164, 25.12310312039844, 993.500033578516], [0, 0, 1, 0], [0, 0, 0, 0], [9E9, 9E9, 9E9, 9E9, 9E9, 9E9]];
    CONST robtarget p3971:= [[1549.7072659187932, 24.838692768471546, 993.500033578516], [0, 0, 1, 0], [0, 0, 0, 0], [9E9, 9E9, 9E9, 9E9, 9E9, 9E9]];
    CONST robtarget p3972:= [[1549.823246837155, 24.621968812418615, 993.500033578516], [0, 0, 1, 0], [0, 0, 0, 0], [9E9, 9E9, 9E9, 9E9, 9E9, 9E9]];
    CONST robtarget p3973:= [[1550.0173503464962, 24.270483306697358, 993.500033578516], [0, 0, 1, 0], [0, 0, 0, 0], [9E9, 9E9, 9E9, 9E9, 9E9, 9E9]];
    CONST robtarget p3974:= [[1550.2323628179183, 23.85774046969871, 993.500033578516], [0, 0, 1, 0], [0, 0, 0, 0], [9E9, 9E9, 9E9, 9E9, 9E9, 9E9]];
    CONST robtarget p3975:= [[1550.4115703773768, 23.48341834731623, 993.500033578516], [0, 0, 1, 0], [0, 0, 0, 0], [9E9, 9E9, 9E9, 9E9, 9E9, 9E9]];
    CONST robtarget p3976:= [[1550.5687657558142, 23.093719493639483, 993.500033578516], [0, 0, 1, 0], [0, 0, 0, 0], [9E9, 9E9, 9E9, 9E9, 9E9, 9E9]];
    CONST robtarget p3977:= [[1550.7708002413533, 22.635993666558633, 993.500033578516], [0, 0, 1, 0], [0, 0, 0, 0], [9E9, 9E9, 9E9, 9E9, 9E9, 9E9]];
    CONST robtarget p3978:= [[1550.8467990254626, 22.455554681534252, 993.500033578516], [0, 0, 1, 0], [0, 0, 0, 0], [9E9, 9E9, 9E9, 9E9, 9E9, 9E9]];
    CONST robtarget p3979:= [[1550.8679927939716, 22.407147495915837, 993.500033578516], [0, 0, 1, 0], [0, 0, 0, 0], [9E9, 9E9, 9E9, 9E9, 9E9, 9E9]];
    CONST robtarget p3980:= [[1551.1782038624883, 21.63213423724774, 993.500033578516], [0, 0, 1, 0], [0, 0, 0, 0], [9E9, 9E9, 9E9, 9E9, 9E9, 9E9]];
    CONST robtarget p3981:= [[1551.3350528787662, 21.314610237893362, 993.500033578516], [0, 0, 1, 0], [0, 0, 0, 0], [9E9, 9E9, 9E9, 9E9, 9E9, 9E9]];
    CONST robtarget p3982:= [[1551.3719342351017, 21.227387124179316, 993.500033578516], [0, 0, 1, 0], [0, 0, 0, 0], [9E9, 9E9, 9E9, 9E9, 9E9, 9E9]];
    CONST robtarget p3983:= [[1551.4393333786395, 21.069937556610597, 993.500033578516], [0, 0, 1, 0], [0, 0, 0, 0], [9E9, 9E9, 9E9, 9E9, 9E9, 9E9]];
    CONST robtarget p3984:= [[1551.560197454426, 20.763500377956504, 993.500033578516], [0, 0, 1, 0], [0, 0, 0, 0], [9E9, 9E9, 9E9, 9E9, 9E9, 9E9]];
    CONST robtarget p3985:= [[1551.668252798264, 20.496177078395547, 993.500033578516], [0, 0, 1, 0], [0, 0, 0, 0], [9E9, 9E9, 9E9, 9E9, 9E9, 9E9]];
    CONST robtarget p3986:= [[1551.702927823328, 20.41695000518267, 993.500033578516], [0, 0, 1, 0], [0, 0, 0, 0], [9E9, 9E9, 9E9, 9E9, 9E9, 9E9]];
    CONST robtarget p3987:= [[1551.9130155821983, 19.938310087453388, 993.500033578516], [0, 0, 1, 0], [0, 0, 0, 0], [9E9, 9E9, 9E9, 9E9, 9E9, 9E9]];
    CONST robtarget p3988:= [[1552.0521719180438, 19.5196678454153, 993.500033578516], [0, 0, 1, 0], [0, 0, 0, 0], [9E9, 9E9, 9E9, 9E9, 9E9, 9E9]];
    CONST robtarget p3989:= [[1552.1514795297917, 19.253582051572337, 993.500033578516], [0, 0, 1, 0], [0, 0, 0, 0], [9E9, 9E9, 9E9, 9E9, 9E9, 9E9]];
    CONST robtarget p3990:= [[1552.2193140653824, 19.0550242267619, 993.500033578516], [0, 0, 1, 0], [0, 0, 0, 0], [9E9, 9E9, 9E9, 9E9, 9E9, 9E9]];
    CONST robtarget p3991:= [[1552.4526656990831, 18.374031272872386, 993.500033578516], [0, 0, 1, 0], [0, 0, 0, 0], [9E9, 9E9, 9E9, 9E9, 9E9, 9E9]];
    CONST robtarget p3992:= [[1552.538204603163, 18.1430395759227, 993.500033578516], [0, 0, 1, 0], [0, 0, 0, 0], [9E9, 9E9, 9E9, 9E9, 9E9, 9E9]];
    CONST robtarget p3993:= [[1552.7201740314629, 17.598178722742034, 993.500033578516], [0, 0, 1, 0], [0, 0, 0, 0], [9E9, 9E9, 9E9, 9E9, 9E9, 9E9]];
    CONST robtarget p3994:= [[1552.855690735831, 17.185623387349494, 993.500033578516], [0, 0, 1, 0], [0, 0, 0, 0], [9E9, 9E9, 9E9, 9E9, 9E9, 9E9]];
    CONST robtarget p3995:= [[1552.9254527924388, 16.968011815428426, 993.500033578516], [0, 0, 1, 0], [0, 0, 0, 0], [9E9, 9E9, 9E9, 9E9, 9E9, 9E9]];
    CONST robtarget p3996:= [[1552.9558504180025, 16.873434373046294, 993.500033578516], [0, 0, 1, 0], [0, 0, 0, 0], [9E9, 9E9, 9E9, 9E9, 9E9, 9E9]];
    CONST robtarget p3997:= [[1553.0879547869743, 16.498579819879424, 993.500033578516], [0, 0, 1, 0], [0, 0, 0, 0], [9E9, 9E9, 9E9, 9E9, 9E9, 9E9]];
    CONST robtarget p3998:= [[1553.261496025404, 16.020898589821982, 993.500033578516], [0, 0, 1, 0], [0, 0, 0, 0], [9E9, 9E9, 9E9, 9E9, 9E9, 9E9]];
    CONST robtarget p3999:= [[1553.3803917591945, 15.549265232169603, 993.500033578516], [0, 0, 1, 0], [0, 0, 0, 0], [9E9, 9E9, 9E9, 9E9, 9E9, 9E9]];
    CONST robtarget p4000:= [[1553.504362419036, 15.085755780383863, 993.500033578516], [0, 0, 1, 0], [0, 0, 0, 0], [9E9, 9E9, 9E9, 9E9, 9E9, 9E9]];
    CONST robtarget p4001:= [[1553.5778545527398, 14.776171116563674, 993.500033578516], [0, 0, 1, 0], [0, 0, 0, 0], [9E9, 9E9, 9E9, 9E9, 9E9, 9E9]];
    CONST robtarget p4002:= [[1553.6491965844975, 14.515382670084577, 993.500033578516], [0, 0, 1, 0], [0, 0, 0, 0], [9E9, 9E9, 9E9, 9E9, 9E9, 9E9]];
    CONST robtarget p4003:= [[1553.667349034861, 14.437207906990423, 993.500033578516], [0, 0, 1, 0], [0, 0, 0, 0], [9E9, 9E9, 9E9, 9E9, 9E9, 9E9]];
    CONST robtarget p4004:= [[1553.8741959168074, 13.674859848647714, 993.500033578516], [0, 0, 1, 0], [0, 0, 0, 0], [9E9, 9E9, 9E9, 9E9, 9E9, 9E9]];
    CONST robtarget p4005:= [[1554.0412050177044, 13.025063242685178, 993.500033578516], [0, 0, 1, 0], [0, 0, 0, 0], [9E9, 9E9, 9E9, 9E9, 9E9, 9E9]];
    CONST robtarget p4006:= [[1554.096687627747, 12.789672785285006, 993.500033578516], [0, 0, 1, 0], [0, 0, 0, 0], [9E9, 9E9, 9E9, 9E9, 9E9, 9E9]];
    CONST robtarget p4007:= [[1554.22540993021, 12.3086575654726, 993.500033578516], [0, 0, 1, 0], [0, 0, 0, 0], [9E9, 9E9, 9E9, 9E9, 9E9, 9E9]];
    CONST robtarget p4008:= [[1554.2411862989752, 12.250140405912376, 993.500033578516], [0, 0, 1, 0], [0, 0, 0, 0], [9E9, 9E9, 9E9, 9E9, 9E9, 9E9]];
    CONST robtarget p4009:= [[1554.2824650031757, 12.099864492202414, 993.500033578516], [0, 0, 1, 0], [0, 0, 0, 0], [9E9, 9E9, 9E9, 9E9, 9E9, 9E9]];
    CONST robtarget p4010:= [[1554.304639486967, 12.00262079639036, 993.500033578516], [0, 0, 1, 0], [0, 0, 0, 0], [9E9, 9E9, 9E9, 9E9, 9E9, 9E9]];
    CONST robtarget p4011:= [[1554.3716911842698, 11.646362812083439, 993.500033578516], [0, 0, 1, 0], [0, 0, 0, 0], [9E9, 9E9, 9E9, 9E9, 9E9, 9E9]];
    CONST robtarget p4012:= [[1554.4582118750636, 11.161584922314006, 993.500033578516], [0, 0, 1, 0], [0, 0, 0, 0], [9E9, 9E9, 9E9, 9E9, 9E9, 9E9]];
    CONST robtarget p4013:= [[1554.4979948302853, 10.891442683281767, 993.500033578516], [0, 0, 1, 0], [0, 0, 0, 0], [9E9, 9E9, 9E9, 9E9, 9E9, 9E9]];
    CONST robtarget p4014:= [[1554.5990339472123, 10.408058462202789, 993.500033578516], [0, 0, 1, 0], [0, 0, 0, 0], [9E9, 9E9, 9E9, 9E9, 9E9, 9E9]];
    CONST robtarget p4015:= [[1554.6061902281515, 10.369215536107092, 993.500033578516], [0, 0, 1, 0], [0, 0, 0, 0], [9E9, 9E9, 9E9, 9E9, 9E9, 9E9]];
